// TwinCAT 3 PLC project TcoCoreExamples
// Title: TcoCoreExamples
// Company: Vortex.Library
// Author: Inxton
// ProjectVersion: 0.6.0.913
// ProgramVersion: 3.1.4024.12
// libraries:
//   Tc2_Standard, * (Beckhoff Automation GmbH)
//   Tc2_System, * (Beckhoff Automation GmbH)
//   Tc3_Module, * (Beckhoff Automation GmbH)
//   TcoCore, 0.6.0.913 (Vortex.Library)
// project tree:
//   Examples/Components/Digital/TcoDi/ TcoDi.TcPOU, TcoDiConfig.TcDUT
//   Examples/Components/Digital/TcoDo/ TcoDo.TcPOU
//   Examples/Components/ fbPiston.TcPOU, fbPistonConfig.TcDUT, fbPistonStatus.TcDUT, fbPistonMoveTask.TcPOU, IPistonGripper.TcIO, IPistonHorizontal.TcIO, IPistonVertical.TcIO
//   Examples/Components/WrappedComponent/ Example1WrappedComponent.TcPOU, Example2WrappedComponent.TcPOU, Example2WrappedComponents.TcDUT, Example2WrappedComponents_Status.TcDUT, Example2WrappedComponents_Config.TcDUT, Example2WrappedComponents_Control.TcDUT
//   Examples/Dialogs/ DiaglogsContext.TcPOU, MyOwnContent.TcPOU
//   Examples/ EXAMPLES_PRG.TcPOU, fbContext.TcPOU
//   Examples/Implementation/TcoContext/ TcoContext_App_1.TcPOU
//   Examples/Implementation/TcoObject/ TcoObject_Counter.TcPOU
//   Examples/Implementation/TcoState/ TcoContext_App_2.TcPOU
//   Examples/Implementation/TcoTask/ TcoTask_DownCounter.TcPOU
//   Examples/Logger/ LoggerContext.TcPOU, LoggerUsage.TcPOU
//   Examples/Manipulator/ fbManipulatorAutomat.TcPOU, fbManipulatorContext.TcPOU, gMANIPULATOR_IO.TcGVL, MANIPULATOR.TcPOU
//   Examples/Recorder/ RecordableStation001.TcPOU, RecordableStation001_Components.TcPOU, RecordableStation001_Sequencer.TcPOU
//   Examples/Station_001/ Station001.TcPOU, Station001_Components.TcPOU, Station001_Sequencer.TcPOU
//   Examples/Station_002/ Station002.TcPOU
//   Examples/Structured/ StructuredData.TcDUT, StructuredObject.TcPOU, StrucuredContext.TcPOU
//   Examples/WaveForm/ eTransitionType.TcDUT, TcoContext_Waveform.TcPOU, TcoObject_Waveform.TcPOU, TcoState_WaveformSequence.TcPOU, TcoTask_Transition.TcPOU, WaveformPoint.TcDUT
//   / PlcTask.TcTTO
//   POUs/ MAIN.TcPOU
// (motion and I/O tree: see PLC project tcocore)
// real-time tasks:
//   TASK PlcTask: cycle T#10ms, priority 20, ADS port 350
//   TASK PlcTask1: cycle T#10ms, priority 21, ADS port 351
//   TASK PlcTask2: cycle T#10ms, priority 22, ADS port 352

CONFIGURATION TcoCoreExamples
    RESOURCE PLC ON TwinCAT3
        TASK PlcTask(INTERVAL := T#10ms, PRIORITY := 22);
        PROGRAM MAIN WITH PlcTask : MAIN;
    END_RESOURCE
END_CONFIGURATION

// ---- Examples/Components/Digital/TcoDi/TcoDiConfig.TcDUT
TYPE TcoDiConfig :
STRUCT
    IsFalseTimeOut : TIME := T#10S;
    IsTrueTimeOut : TIME := T#10S;
END_STRUCT
END_TYPE

// ---- Examples/Components/fbPistonConfig.TcDUT
TYPE fbPistonConfig :
STRUCT
    MaxTimeToReachHome : TIME;
    MaxTimeToReachWork : TIME;
END_STRUCT
END_TYPE

// ---- Examples/Components/fbPistonStatus.TcDUT
TYPE fbPistonStatus :
STRUCT
    AtHome : TIME;
    AtWork : TIME;
END_STRUCT
END_TYPE

// ---- Examples/Components/WrappedComponent/Example2WrappedComponents.TcDUT
TYPE Example2WrappedComponents EXTENDS TcoCore.TcoStruct :
STRUCT
    {attribute addProperty Name "Pneumatic cyclinder"}
    piston : fbPiston(THISSTRUCT);
    digitalInput : TcoDi(THISSTRUCT);
    digitaOutput : TcoDo(THISSTRUCT);
    dummy1Task : TcoCore.TcoTask(THISSTRUCT);
    dummy2Task : TcoCore.TcoTask(THISSTRUCT);
    Setpoint : INT;
END_STRUCT
END_TYPE

// ---- Examples/Components/WrappedComponent/Example2WrappedComponents_Status.TcDUT
TYPE Example2WrappedComponents_Status EXTENDS TcoCore.TcoStruct :
STRUCT
    Feedback1 : INT;
    Feedback2 : BOOL;
    Feedback3 : STRING;
END_STRUCT
END_TYPE

// ---- Examples/Components/WrappedComponent/Example2WrappedComponents_Config.TcDUT
TYPE Example2WrappedComponents_Config EXTENDS TcoCore.TcoStruct :
STRUCT
    Setpoint1 : INT;
    Active : BOOL;
    FeedbackRequest : STRING;
END_STRUCT
END_TYPE

// ---- Examples/Components/WrappedComponent/Example2WrappedComponents_Control.TcDUT
TYPE Example2WrappedComponents_Control EXTENDS TcoCore.TcoStruct :
STRUCT
    Setpoint1 : INT;
    Up : BOOL;
    CommandAscii : STRING;
END_STRUCT
END_TYPE

// ---- Examples/Structured/StructuredData.TcDUT
TYPE StructuredData EXTENDS TcoCore.TcoStruct :
STRUCT
    _o1 :
STRUCTuredObject(THISSTRUCT);
END_STRUCT
END_TYPE

// ---- Examples/WaveForm/eTransitionType.TcDUT
{attribute 'qualified_only'}
{attribute 'strict'}
TYPE eTransitionType :
(
    None := 0,
    Linear := 1,
    Exponential := 2,
    S_Type := 3
);
END_TYPE

// ---- Examples/WaveForm/WaveformPoint.TcDUT
TYPE WaveformPoint :
STRUCT
    TransitionType : eTransitionType;
    TargetValue : LREAL; //Value to be reached in "Duration" PLC cycles
    Duration : UINT; //Number of PLC cycles during which the "TargetValue" must be reached
    Shape : LREAL; //Define curve shape
END_STRUCT
END_TYPE

// ---- Examples/Manipulator/gMANIPULATOR_IO.TcGVL
{attribute 'qualified_only'}
VAR_GLOBAL
    Inputs AT %I* : ARRAY[0..7] OF BOOL;
    Outputs AT %Q* : ARRAY[0..7] OF BOOL;
END_VAR

// ---- Examples/Components/IPistonGripper.TcIO
INTERFACE IPistonGripper

METHOD Close : TcoCore.ITcoTaskStatus
END_METHOD

METHOD Open : TcoCore.ITcoTaskStatus
END_METHOD

END_INTERFACE

// ---- Examples/Components/IPistonHorizontal.TcIO
INTERFACE IPistonHorizontal

METHOD MoveLeft : TcoCore.ITcoTaskStatus
END_METHOD

METHOD MoveRight : TcoCore.ITcoTaskStatus
END_METHOD

END_INTERFACE

// ---- Examples/Components/IPistonVertical.TcIO
INTERFACE IPistonVertical

METHOD MoveDown : TcoCore.ITcoTaskStatus
END_METHOD

METHOD MoveUp : TcoCore.ITcoTaskStatus
END_METHOD

END_INTERFACE

// ---- POUs/MAIN.TcPOU
PROGRAM MAIN
VAR
    _station001 : Station001;
    _station002 : Station002;
END_VAR

EXAMPLES_PRG();
MANIPULATOR();
_station001._sequence.DeactivateDeveloperChecks();
_station001.Run();
_station002.Run();

END_PROGRAM

// ---- Examples/Station_001/Station001.TcPOU
FUNCTION_BLOCK Station001 EXTENDS TcoCore.TcoContext
VAR
    {attribute addProperty Name "Long running example"}
    LongRunningTask : TcoCore.TcoTask(THIS^);
    i : int;
    _components : Station001_Components(THIS^);
    _sequence : Station001_Sequencer(THIS^, eRestoreMode.None, _components);
END_VAR

(*~
    <docu>
        <summary>
            Main method of the TcoContext. This is the entry point of any control logic that belongs to this context.
            The call of this method is ensured by calling the <c>InstanceName.Run()</c> method, and it must not be called explicitly.
            This method is abstract, and it must be overridden in derived block.
        </summary>
    </docu>
~*)
METHOD PROTECTED Main
_sequence.Run();

IF (LongRunningTask.Execute()) THEN
    i := i + 1;

    IF (i MOD 2000 = 0) THEN
        i := 1;
        LongRunningTask.DoneWhen(TRUE);
    END_IF
END_IF
END_METHOD

END_FUNCTION_BLOCK

// ---- Examples/Station_001/Station001_Components.TcPOU
FUNCTION_BLOCK Station001_Components EXTENDS TcoCore.TcoObject
VAR
    {attribute addProperty Name "Horizontal cyclinder A1"}
    _horizontal : fbPiston(THIS^);
    {attribute addProperty Name "Vertical cyclinder A2"}
    _vertical : fbPiston(THIS^);
    {attribute addProperty Name "Gripper A3"}
    _gripper : fbPiston(THIS^);
    {attribute addProperty Name "Digital input"}
    _di : TcoDi(THIS^);
    {attribute addProperty Name "Wrapped component example 1"}
    _wrappedComponent1 : Example1WrappedComponent(THIS^);
    {attribute addProperty Name "Wrapped component example 2"}
    _wrappedComponent2 : Example2WrappedComponent(THIS^);
    {attribute clr [RenderIgnore()]}
    _wrappedComponents : Example2WrappedComponents;
    tempSisgnal : BOOL;
    temp2Sisgnal : BOOL;
END_VAR
VAR
    _simTimerValue : UINT := 500;
    _simTimer : Tc2_Standard.TON;
END_VAR

_vertical();
_vertical.Service();
_horizontal();
_horizontal.Service();
_gripper();
_wrappedComponent1(inSignal := tempSisgnal);
_wrappedComponent1.Service();
_wrappedComponent2.Components.digitalInput(inoSignal := tempSisgnal);
_wrappedComponent2.Components.digitaOutput(inoSignal := temp2Sisgnal);
_wrappedComponent2();
_wrappedComponent2.Service();
_simTimer(IN := TRUE, PT := UINT_TO_TIME(_simTimerValue));
SimulateCylinder(_vertical);
SimulateCylinder(_horizontal);
SimulateCylinder(_gripper);

PROPERTY Gripper : IPistonGripper
GET
Gripper := _gripper;
END_GET
END_PROPERTY

PROPERTY Horizontal : IPistonHorizontal
GET
Horizontal := _horizontal;
END_GET
END_PROPERTY

METHOD SimulateCylinder
VAR_IN_OUT
    ioCyclinder : fbPiston;
END_VAR
ioCyclinder.iHomePositionSensor := ioCyclinder.qHomePositionActuator AND _simTimer.Q;
ioCyclinder.iWorkPositionSensor := ioCyclinder.qWorkPositionActuator AND _simTimer.Q;
END_METHOD

PROPERTY Vertical : IPistonVertical
GET
Vertical := _vertical;
END_GET
END_PROPERTY

END_FUNCTION_BLOCK

// ---- Examples/Components/fbPiston.TcPOU
{attribute addProperty Name "Pneumatic cyclinder"}
FUNCTION_BLOCK fbPiston EXTENDS TcoCore.TcoComponent IMPLEMENTS IPistonGripper, IPistonHorizontal, IPistonVertical
VAR_INPUT
    iHomePositionSensor : BOOL;
    iWorkPositionSensor : BOOL;
END_VAR
VAR_OUTPUT
    qHomePositionActuator : BOOL;
    qWorkPositionActuator : BOOL;
END_VAR
VAR
    {attribute addProperty Activity "moves to home position"}
    _moveHomeTask : fbPistonMoveTask(THIS^);
    {attribute addProperty Activity "moves to work position"}
    _moveWorkTask : fbPistonMoveTask(THIS^);
    _moveHomeMomentaryTask : TcoCore.TcoMomentaryTask(THIS^);
    _moveHomeToggleTask : TcoCore.TcoToggleTask(THIS^, FALSE);
    _config : fbPistonConfig;
    _status : fbPistonStatus;
END_VAR

_moveHomeTask(PositionSensor := iHomePositionSensor, MoveToPositionSignal := qHomePositionActuator, InverseSignal := qWorkPositionActuator);
_moveWorkTask(PositionSensor := iWorkPositionSensor, MoveToPositionSignal := qWorkPositionActuator, InverseSignal := qHomePositionActuator);
_moveHomeMomentaryTask.Run();
_moveHomeToggleTask.Toggle();

METHOD Close : TcoCore.ITcoTaskStatus
Close := MoveToHome();
END_METHOD

METHOD MoveDown : TcoCore.ITcoTaskStatus
MoveDown := MoveToHome();
END_METHOD

METHOD MoveLeft : TcoCore.ITcoTaskStatus
MoveLeft := MoveToWork();
END_METHOD

METHOD MoveRight : TcoCore.ITcoTaskStatus
MoveRight := MoveToHome();
END_METHOD

METHOD PROTECTED MoveToHome : TcoCore.ITcoTaskStatus
MoveToHome := THIS^._moveHomeTask.Invoke();
END_METHOD

METHOD PROTECTED MoveToWork : TcoCore.ITcoTaskStatus
MoveToWork := THIS^._moveWorkTask.Invoke();
END_METHOD

METHOD MoveUp : TcoCore.ITcoTaskStatus
MoveUp := MoveToWork();
END_METHOD

METHOD Open : TcoCore.ITcoTaskStatus
Open := MoveToWork();
END_METHOD

METHOD Restore : ITcoRestorable
THIS^._moveHomeTask.Restore();
THIS^._moveWorkTask.Restore();
END_METHOD

(*~
    <docu>
        <summary>
            Custom service (manual, maintenance) logic.
            This method must be implemented in derived class.
        </summary>
    </docu>
~*)
METHOD PROTECTED ServiceMode
END_METHOD

END_FUNCTION_BLOCK

// ---- Examples/Components/fbPistonMoveTask.TcPOU
{attribute addProperty Activity "task is running"}
FUNCTION_BLOCK fbPistonMoveTask EXTENDS TcoCore.TcoTask
VAR_INPUT
    PositionSensor : BOOL;
END_VAR
VAR_IN_OUT
    MoveToPositionSignal : BOOL;
    InverseSignal : BOOL;
END_VAR

IF (THIS^.Execute()) THEN
    THIS^.Messenger.Debug('|[[1]AttributeName]| |[AttributeActivity]|, extremity sensor not reached yet.');
    InverseSignal := FALSE;
    MoveToPositionSignal := TRUE;
    ThrowWhen(THIS^.ElapsedTime > T#5S);
    THIS^.DoneWhen(PositionSensor);
END_IF

END_FUNCTION_BLOCK

// ---- Examples/Components/Digital/TcoDi/TcoDi.TcPOU
(*~
    <docu>
        <summary>
                Generic component for monitoring of an input. (e.g. DigitalSensor).
        </summary>
    </docu>
~*)
FUNCTION_BLOCK TcoDi EXTENDS TcoCore.TcoComponent
VAR_IN_OUT
    (*~
    <docu>
        <summary>
            Input signal. Typically an `%I*` variable.
        </summary>
    </docu>
    ~*)
    inoSignal : BOOL;
END_VAR
VAR
    (*~
    <docu>
        <summary>
            Backing variable for signal; this variable is used directly by the component. It updates `inoSingal` in FB body call.
        </summary>
    </docu>
    ~*)
    _signal : BOOL;
END_VAR
VAR
    {attribute addProperty Name "<#Signal#>"}
    _signalInfo : TcoCore.TcoSignalInfo;
    {attribute addProperty Name "<#Check On#>"}
    {attribute addProperty ToolTip "<#Checks that the input is on#>"}
    _isTrueTask : TcoCore.TcoTask(THIS^);
    {attribute addProperty ToolTip "<#Checks that the input is off#>"}
    {attribute addProperty Name "<#Check Off#>"}
    _isFalseTask : TcoCore.TcoTask(THIS^);
    _config : TcoDiConfig;
    _isFalseTimeOutTimers : Tc2_Standard.TON;
    _isTrueTimeOutTimers : Tc2_Standard.TON;
END_VAR

IF (__ISVALIDREF(inoSignal)) THEN
    _signalInfo.GetSignalInfo(SIZEOF(inoSignal), ADR(inoSignal));
    _signal := inoSignal;
END_IF;

IF (_isTrueTask.Execute()) THEN
    _isTrueTask.DoneWhen(IsTrue);
END_IF

IF (_isFalseTask.Execute()) THEN
    _isFalseTask.DoneWhen(IsFalse);
END_IF

PROPERTY Config : REFERENCE TO TcoDiConfig
GET
Config REF= _config;
END_GET
END_PROPERTY

METHOD FB_init : BOOL
VAR_INPUT
    bInitRetains : BOOL; // if TRUE, the retain variables are initialized (warm start / cold start)
    bInCopyCode : BOOL; // if TRUE, the instance afterwards gets moved into the copy code (online change)
    ParentObject : ITcoObject;
END_VAR
END_METHOD

(*~
    <docu>
        <summary>
            Gets 'true' when monitor signal is 'off/false/logical 0'.
            Generates message when the returning 'false'.
        </summary>
    </docu>
~*)
{attribute 'monitoring' := 'variable'}
PROPERTY IsFalse : BOOL
GET
IsFalse := NOT _signal;
_isFalseTimeOutTimers(IN := NOT IsFalse, PT := _config.IsFalseTimeOut);

IF (NOT IsFalse) THEN
    Messenger.Info('<#Expecting `negative` signal#>');
END_IF;

IF (_isFalseTimeOutTimers.Q) THEN
    Messenger.Warning('<#Expecting `negative` signal#>');
END_IF;
END_GET
END_PROPERTY

(*~
    <docu>
        <summary>
            Gets 'true' when monitor signal is 'on/true/logical 1'.
            Generates message when the returning 'false'.
        </summary>
    </docu>
~*)
{attribute 'monitoring' := 'variable'}
PROPERTY IsTrue : BOOL
GET
IsTrue := _signal;
_isTrueTimeOutTimers(IN := NOT IsTrue, PT := _config.IsFalseTimeOut);

IF (NOT IsTrue) THEN
    Messenger.Info('<#Expecting `positive` signal#>');
END_IF;

IF (_isTrueTimeOutTimers.Q) THEN
    Messenger.Warning('<#Expecting `positive` signal#>');
END_IF;
END_GET
END_PROPERTY

(*~
    <docu>
        <summary>
            Restores this instance to the Ready state. Can be called explicitly or from within one of the restore mechanisms.
        </summary>
    </docu>
~*)
METHOD Restore : ITcoRestorable
// No implementation needed for this componet.
END_METHOD

(*~
    <docu>
        <summary>
            Custom service (manual, maintenance) logic.
            This method must be implemented in derived class.
        </summary>
    </docu>
~*)
METHOD PROTECTED ServiceMode
END_METHOD

PROPERTY PUBLIC Signal : Bool
GET
Signal := _signal;
END_GET
END_PROPERTY

END_FUNCTION_BLOCK

// ---- Examples/Components/WrappedComponent/Example1WrappedComponent.TcPOU
FUNCTION_BLOCK Example1WrappedComponent EXTENDS TcoCore.TcoComponent
VAR_INPUT
    inSignal : BOOL;
END_VAR
VAR_OUTPUT
END_VAR
VAR
    piston : fbPiston(THIS^);
    digitalInput : TcoDi(THIS^);
    digitaOutput : TcoDo(THIS^);
    dummy1Task : TcoCore.TcoTask(THIS^);
    dummy2Task : TcoCore.TcoTask(THIS^);
    Setpoint : INT;
END_VAR

piston();
digitalInput(inoSignal := inSignal);
dummy1Task.Enabled := TRUE;

IF dummy1Task.Execute() THEN
    ;
END_IF

(*~
    <docu>
        <summary>
            Restores this instance to the Ready state. Can be called explicitly or from within one of the restore mechanisms.
        </summary>
    </docu>
~*)
METHOD Restore : ITcoRestorable
END_METHOD

(*~
    <docu>
        <summary>
            Custom service (manual, maintenance) logic.
            This method must be implemented in derived class.
        </summary>
    </docu>
~*)
METHOD PROTECTED ServiceMode
piston.Service();
digitalInput.Service();
digitaOutput.Service();
END_METHOD

END_FUNCTION_BLOCK

// ---- Examples/Components/Digital/TcoDo/TcoDo.TcPOU
(*~
    <docu>
        <summary>
                Generic component for discrete control of an output.
        </summary>
    </docu>
~*)
FUNCTION_BLOCK TcoDo EXTENDS TcoCore.TcoComponent
VAR_IN_OUT
    (*~
    <docu>
        <summary>
            Controlled signal. Typically an `%Q*` variable.
        </summary>
    </docu>
    ~*)
    inoSignal : BOOL;
END_VAR
VAR
    (*~
    <docu>
        <summary>
            Backing variable for signal; this variable is used directly by the component. It updates `inoSingal` in FB body call.
        </summary>
    </docu>
    ~*)
    _signal : BOOL;
END_VAR
VAR
    {attribute addProperty Name "<#Signal#>"}
    _signalInfo : TcoCore.TcoSignalInfo;
    {attribute addProperty Name "<#On#>"}
    {attribute addProperty ToolTip "<#Sets the output#>"}
    _setTask : TcoCore.TcoTask(THIS^);
    {attribute addProperty ToolTip "<#Resets the output#>"}
    {attribute addProperty Name "<#Off#>"}
    _resetTask : TcoCore.TcoTask(THIS^);
END_VAR

IF (__ISVALIDREF(inoSignal)) THEN
    _signalInfo.GetSignalInfo(SIZEOF(inoSignal), ADR(inoSignal));
    inoSignal := _signal;
END_IF;

IF (_setTask.Execute()) THEN
    _setTask.DoneWhen(Set());
END_IF

IF (_resetTask.Execute()) THEN
    _resetTask.DoneWhen(Reset());
END_IF

METHOD FB_init : BOOL
VAR_INPUT
    bInitRetains : BOOL; // if TRUE, the retain variables are initialized (warm start / cold start)
    bInCopyCode : BOOL; // if TRUE, the instance afterwards gets moved into the copy code (online change)
    ParentObject : ITcoObject;
END_VAR
END_METHOD

(*~
    <docu>
        <summary>
            Gets 'true' when monitor signal is 'off/false/logical 0'.
            Generates message when the returning 'false'.
        </summary>
    </docu>
~*)
{attribute 'monitoring' := 'variable'}
PROPERTY IsFalse : BOOL
GET
IsFalse := NOT _signal;

IF (NOT IsFalse) THEN
    Messenger.Info('<#Expecting `negative` signal#>');
END_IF;
END_GET
END_PROPERTY

(*~
    <docu>
        <summary>
            Gets 'true' when monitor signal is 'on/true/logical 1'.
            Generates message when the returning 'false'.
        </summary>
    </docu>
~*)
{attribute 'monitoring' := 'variable'}
PROPERTY IsTrue : BOOL
GET
IsTrue := _signal;

IF (NOT IsTrue) THEN
    Messenger.Info('<#Expecting `positive` signal#>');
END_IF;
END_GET
END_PROPERTY

(*~
    <docu>
        <summary>
            Sets controlled signal into 'off/false/logical 0'.
        </summary>
    </docu>
~*)
METHOD Reset : BOOL
Messenger.Trace('<#Reseting signal (off/false)#>');
_signal := FALSE;
Reset := TRUE;
END_METHOD

(*~
    <docu>
        <summary>
            Restores this instance to the Ready state. Can be called explicitly or from within one of the restore mechanisms.
        </summary>
    </docu>
~*)
METHOD Restore : ITcoRestorable
// No implementation needed for this componet.
END_METHOD

(*~
    <docu>
        <summary>
            Custom service (manual, maintenance) logic.
            This method must be implemented in derived class.
        </summary>
    </docu>
~*)
METHOD PROTECTED ServiceMode
END_METHOD

(*~
    <docu>
        <summary>
            Sets controlled signal into 'on/true/logical 1'.
        </summary>
    </docu>
~*)
METHOD PUBLIC Set : BOOL
Messenger.Trace('<#Setting signal (on/true)#>');
_signal := TRUE;
Set := TRUE;
END_METHOD

PROPERTY PUBLIC Signal : Bool
GET
Signal := _signal;
END_GET
END_PROPERTY

END_FUNCTION_BLOCK

// ---- Examples/Components/WrappedComponent/Example2WrappedComponent.TcPOU
FUNCTION_BLOCK Example2WrappedComponent EXTENDS TcoCore.TcoComponent
VAR_OUTPUT
END_VAR
VAR
    _config : Example2WrappedComponents_Config;
    _status : Example2WrappedComponents_Status;
    _control : Example2WrappedComponents_Control;
    _components : Example2WrappedComponents := (Parent := THIS^);
    _resetTask : TcoCore.TcoTask(THIS^);
    _restoreTask : TcoCore.TcoTask(THIS^);
    Setpoint : INT;
    {attribute clr [RenderIgnore()]}
    SetpointDoNotRender : INT;
END_VAR

_resetTask();

PROPERTY Components : REFERENCE TO Example2WrappedComponents
GET
Components ref= _components;
END_GET
END_PROPERTY

(*~
    <docu>
        <summary>
            Restores this instance to the Ready state. Can be called explicitly or from within one of the restore mechanisms.
        </summary>
    </docu>
~*)
METHOD Restore : ITcoRestorable
END_METHOD

(*~
    <docu>
        <summary>
            Custom service (manual, maintenance) logic.
            This method must be implemented in derived class.
        </summary>
    </docu>
~*)
METHOD PROTECTED ServiceMode
_components.piston.Service();
_components.digitalInput.Service();
_components.digitaOutput.Service();
END_METHOD

END_FUNCTION_BLOCK

// ---- Examples/Station_001/Station001_Sequencer.TcPOU
FUNCTION_BLOCK Station001_Sequencer EXTENDS TcoCore.TcoSequencer
VAR
    components : REFERENCE TO Station001_Components;
END_VAR
VAR
    _switchToStep : BOOL;
    _failedToLoad : BOOL;
END_VAR
VAR
    _onStateChangeCount : LREAL;
    _sequenceCompleteCount : LREAL;
    _stepsPerSequence : LREAL;
END_VAR
VAR
    _stepIdChange : INT := 400;
    _stepsCountChange : BOOL := FALSE;
END_VAR

METHOD FB_init : BOOL
VAR_INPUT
    bInitRetains : BOOL; // if TRUE, the retain variables are initialized (warm start / cold start)
    bInCopyCode : BOOL; // if TRUE, the instance afterwards gets moved into the copy code (online change)
    ParentObject : ITcoObject;
    AutoRestoreMode : eRestoreMode;
    refComponents : REFERENCE TO Station001_Components;
END_VAR
Components REF= refComponents;
END_METHOD

METHOD Init
VAR_INPUT
END_VAR
components();
END_METHOD

(*~
    <docu>
        <summary>
            Main method of the sequener. Custom code needs to be placed here. The sequencer is executed by call of InstanceName.Run() method.
            This method is abstract, and it must be overridden in derived block.
        </summary>
    </docu>
~*)
METHOD PROTECTED Main : BOOL
Init();
THIS^.Messenger.Info('Stations one sequencer is running.');

IF (Step(100, TRUE, 'MOVE ALL CYLINDERS TO GROUND POSITION')) THEN
    //-----------------------------------------------------
    StepCompleteWhen(components.Vertical.MoveUp().Done AND_THEN components.Horizontal.MoveLeft().Done AND_THEN components.Gripper.Open().Done);
    //-----------------------------------------------------
END_IF

IF (Step(200, TRUE, 'MOVE VERTICAL CYLINDER DOWN')) THEN
    //-----------------------------------------------------
    StepCompleteWhen(components.Vertical.MoveDown().Done);
    //-----------------------------------------------------
END_IF

IF NOT _stepsCountChange THEN
    IF (Step(300, TRUE, 'CLOSE GRIPPER')) THEN
        //-----------------------------------------------------
        IF (components.Gripper.Close().Done) THEN
            IF (_failedToLoad) THEN
                RequestStep(100);
            ELSE
                StepCompleteWhen(TRUE);
            END_IF;
        END_IF;
        //-----------------------------------------------------
    END_IF

    IF (Step(_stepIdChange, TRUE, 'MOVE VERTICAL CYLINDER UP')) THEN
        //-----------------------------------------------------
        StepCompleteWhen(components.Vertical.MoveUp().Done);
        //-----------------------------------------------------
    END_IF

    IF (Step(500, TRUE, 'MOVE HORIZONTAL CYLINDER TO UNLOAD POSITION')) THEN
        //-----------------------------------------------------
        StepCompleteWhen(components.Horizontal.MoveRight().Done);
        //-----------------------------------------------------
    END_IF
END_IF

IF (Step(600, TRUE, 'MOVE VERTICAL CYLINDER DOWN')) THEN
    //-----------------------------------------------------
    StepCompleteWhen(components.Vertical.MoveDown().Done);
    //-----------------------------------------------------
END_IF

IF (Step(700, TRUE, 'OPEN GRIPPER')) THEN
    //-----------------------------------------------------
    StepCompleteWhen(components.Gripper.Open().Done);
    //-----------------------------------------------------
END_IF

IF (Step(800, TRUE, 'CLOSE SEQUENCE')) THEN
    //-----------------------------------------------------
    _sequenceCompleteCount := _sequenceCompleteCount + 1;
    _stepsPerSequence := (_onStateChangeCount - _sequenceCompleteCount + 1) / _sequenceCompleteCount;
    CompleteSequence();
    //-----------------------------------------------------
END_IF

THIS^.Messenger.Debug('THIS IS DEBUG DIAG MESSAGE ');
THIS^.Messenger.Info('THIS IS INFO DIAG MESSAGE ');
THIS^.Messenger.Notify('THIS IS NOTIFY DIAG MESSAGE ');
THIS^.Messenger.Warning('THIS IS WARNING DIAG MESSAGE ');
//THIS^.Messenger.Error('THIS IS ERROR DIAG MESSAGE ');
//THIS^.Messenger.Programming('THIS IS PROGRAMMING DIAG MESSAGE ');
//THIS^.Messenger.Post('THIS IS Fatal DIAG MESSAGE ', eMessageCategory.Fatal);
//THIS^.Messenger.Post('THIS IS Critical DIAG MESSAGE ', eMessageCategory.Critical);
//THIS^.Messenger.Post('THIS IS Catastrophic DIAG MESSAGE ', eMessageCategory.Catastrophic);
THIS^.Messenger.Trace('THIS IS INFO DIAG MESSAGE ');
END_METHOD

METHOD PROTECTED OnStateChange
VAR_INPUT
    PreviousState : INT;
    NewState : INT;
END_VAR
VAR
    sb : TcoCore.StringBuilder;
END_VAR
THIS^.Messenger.Trace(INT_TO_STRING(PreviousState));
_onStateChangeCount := _onStateChangeCount + 1;
components._simTimer(IN := FALSE);
END_METHOD

END_FUNCTION_BLOCK

// ---- Examples/Station_002/Station002.TcPOU
FUNCTION_BLOCK Station002 EXTENDS TcoCore.TcoContext
VAR
    {attribute addProperty Name "Horizontal cyclinder A1"}
    _horizontal : fbPiston(THIS^);
    {attribute addProperty Name "Vertical cyclinder A2"}
    _vertical : fbPiston(THIS^);
    {attribute addProperty Name "Gripper A3"}
    _gripper : fbPiston(THIS^);
END_VAR
VAR
    _s : TcoCore.TcoSequence(THIS^, eRestoreMode.None);
    _sObserver : TcoCore.TcoSequencerObserver(THIS^);
    _failedToLoad : BOOL;
END_VAR

(*~
    <docu>
        <summary>
            Main method of the TcoContext. This is the entry point of any control logic that belongs to this context.
            The call of this method is ensured by calling the <c>InstanceName.Run()</c> method, and it must not be called explicitly.
            This method is abstract, and it must be overridden in derived block.
        </summary>
    </docu>
~*)
METHOD PROTECTED Main
_s.Open();
THIS^._s.Observer := _sObserver;
THIS^._s.Messenger.Info('Stations two sequencer is running.');

IF (_s.Step(100, TRUE, 'MOVE ALL CYLINDERS TO GROUND POSITION')) THEN
    //-----------------------------------------------------
    _s.StepCompleteWhen(_vertical.MoveUp().Done AND_THEN _horizontal.MoveLeft().Done AND_THEN _gripper.Open().Done);
    //-----------------------------------------------------
END_IF

IF (_s.Step(200, TRUE, 'MOVE VERTICAL CYLINDER DOWN')) THEN
    //-----------------------------------------------------
    _s.StepCompleteWhen(_vertical.MoveDown().Done);
    //-----------------------------------------------------
END_IF

IF (_s.Step(300, TRUE, 'CLOSE GRIPPER')) THEN
    //-----------------------------------------------------
    IF (_gripper.Close().Done) THEN
        IF (_failedToLoad) THEN
            _s.RequestStep(100);
        ELSE
            _s.StepCompleteWhen(TRUE);
        END_IF;
    END_IF;
    //-----------------------------------------------------
END_IF

IF (_s.Step(400, TRUE, 'MOVE VERTICAL CYLINDER UP')) THEN
    //-----------------------------------------------------
    _s.StepCompleteWhen(_vertical.MoveUp().Done);
    //-----------------------------------------------------
END_IF

IF (_s.Step(500, TRUE, 'MOVE HORIZONTAL CYLINDER TO UNLOAD POSITION')) THEN
    //-----------------------------------------------------
    _s.StepCompleteWhen(_horizontal.MoveRight().Done);
    //-----------------------------------------------------
END_IF

IF (_s.Step(600, TRUE, 'MOVE VERTICAL CYLINDER DOWN')) THEN
    //-----------------------------------------------------
    _s.StepCompleteWhen(_vertical.MoveDown().Done);
    //-----------------------------------------------------
END_IF

IF (_s.Step(700, TRUE, 'OPEN GRIPPER')) THEN
    //-----------------------------------------------------
    _s.StepCompleteWhen(_gripper.Open().Done);
    //-----------------------------------------------------
END_IF

IF (_s.Step(800, TRUE, 'CLOSE SEQUENCE')) THEN
    //-----------------------------------------------------
    _s.CompleteSequence();
    //-----------------------------------------------------
END_IF

_s.Close();
END_METHOD

END_FUNCTION_BLOCK

// ---- Examples/EXAMPLES_PRG.TcPOU
PROGRAM EXAMPLES_PRG
VAR
    _context : fbContext;
    _recordableStations : RecordableStation001;
    _loggerContext : LoggerContext;
    _strucuredContext : StrucuredContext;
    _diaglogsContext : DiaglogsContext;
    a : TcoCore.ITcoObject;
END_VAR

_context.Run();
_recordableStations.Run();
_loggerContext.Run();
_diaglogsContext.Run();
a := _strucuredContext._structuredData._o1.Parent;

END_PROGRAM

// ---- Examples/fbContext.TcPOU
FUNCTION_BLOCK fbContext EXTENDS TcoCore.TcoContext
VAR
    {attribute addProperty Name "Toggle task example"}
    {attribute addProperty StateOnDesc "<#Enabled#>"}
    {attribute addProperty StateOffDesc "<#Disabled#>"}
    _toggleTaskExample : TcoCore.TcoToggleTask(THIS^, FALSE);
    {attribute addProperty Name "Momentary task example"}
    {attribute addProperty StateOnDesc "<#Running#>"}
    {attribute addProperty StateOffDesc "<#Stopped#>"}
    _momentaryTaskExample : TcoCore.TcoMomentaryTask(THIS^);
END_VAR

METHOD PROTECTED Main
_toggleTaskExample.Run();
_momentaryTaskExample.Run();
END_METHOD

END_FUNCTION_BLOCK

// ---- Examples/Recorder/RecordableStation001.TcPOU
FUNCTION_BLOCK RecordableStation001 EXTENDS TcoCore.TcoContext
VAR
    _components : RecordableStation001_Components(THIS^);
    _sequence : RecordableStation001_Sequencer(THIS^, eRestoreMode.None);
    _serviceModeTask : TcoCore.TcoTask(THIS^);
    _automatModeTask : TcoCore.TcoTask(THIS^);
END_VAR

(*~
    <docu>
        <summary>
            Main method of the TcoContext. This is the entry point of any control logic that belongs to this context.
            The call of this method is ensured by calling the <c>InstanceName.Run()</c> method, and it must not be called explicitly.
            This method is abstract, and it must be overridden in derived block.
        </summary>
    </docu>
~*)
METHOD PROTECTED Main
_sequence(components := _components);
_components();

IF (_serviceModeTask.Execute()) THEN
    _automatModeTask.Restore();
    _components.Service();
END_IF;

IF (_automatModeTask.Execute()) THEN
    _serviceModeTask.Restore();
    _sequence.Run();
END_IF;
END_METHOD

END_FUNCTION_BLOCK

// ---- Examples/Recorder/RecordableStation001_Components.TcPOU
FUNCTION_BLOCK RecordableStation001_Components EXTENDS TcoCore.TcoObject
VAR
    {attribute addProperty Name "Horizontal cyclinder A1"}
    _horizontal : fbPiston(THIS^);
    {attribute addProperty Name "Vertical cyclinder A2"}
    _vertical : fbPiston(THIS^);
    {attribute addProperty Name "Gripper A3"}
    _gripper : fbPiston(THIS^);
END_VAR
VAR
    _simTimerValue : UINT := 500;
    _simTimer : Tc2_Standard.TON;
END_VAR

_vertical();
_horizontal();
_gripper();

PROPERTY Gripper : IPistonGripper
GET
Gripper := _gripper;
END_GET
END_PROPERTY

PROPERTY Horizontal : IPistonHorizontal
GET
Horizontal := _horizontal;
END_GET
END_PROPERTY

METHOD Service
VAR_INPUT
END_VAR
THIS^._gripper.Service();
THIS^._horizontal.Service();
THIS^._vertical.Service();
END_METHOD

PROPERTY Vertical : IPistonVertical
GET
Vertical := _vertical;
END_GET
END_PROPERTY

END_FUNCTION_BLOCK

// ---- Examples/Recorder/RecordableStation001_Sequencer.TcPOU
FUNCTION_BLOCK RecordableStation001_Sequencer EXTENDS TcoCore.TcoSequencer
VAR_IN_OUT
    components : RecordableStation001_Components;
END_VAR
VAR
    _switchToStep : BOOL;
    _failedToLoad : BOOL;
END_VAR
VAR
    _onStateChangeCount : LREAL;
    _sequenceCompleteCount : LREAL;
    _stepsPerSequence : LREAL;
END_VAR

METHOD FB_init : BOOL
VAR_INPUT
    bInitRetains : BOOL; // if TRUE, the retain variables are initialized (warm start / cold start)
    bInCopyCode : BOOL; // if TRUE, the instance afterwards gets moved into the copy code (online change)
    ParentObject : ITcoObject;
    AutoRestoreMode : eRestoreMode;
END_VAR
END_METHOD

METHOD Init
VAR_INPUT
END_VAR
components();
END_METHOD

(*~
    <docu>
        <summary>
            Main method of the sequener. Custom code needs to be placed here. The sequencer is executed by call of InstanceName.Run() method.
            This method is abstract, and it must be overridden in derived block.
        </summary>
    </docu>
~*)
METHOD PROTECTED Main : BOOL
Init();

IF Step(10, TRUE, 'EXAMPLES_PRG._recordableStations._components._horizontal._moveHomeTask') THEN
    //-------------------------------------------------------
    IF (EXAMPLES_PRG._recordableStations._components._horizontal._moveHomeTask.Invoke().Done) THEN
        StepCompleteWhen(TRUE);
    END_IF;
    //-------------------------------------------------------
END_IF;

IF Step(20, TRUE, 'EXAMPLES_PRG._recordableStations._components._vertical._moveHomeTask') THEN
    //-------------------------------------------------------
    IF (EXAMPLES_PRG._recordableStations._components._vertical._moveHomeTask.Invoke().Done) THEN
        StepCompleteWhen(TRUE);
    END_IF;
    //-------------------------------------------------------
END_IF;

IF Step(30, TRUE, 'EXAMPLES_PRG._recordableStations._components._gripper._moveHomeTask') THEN
    //-------------------------------------------------------
    IF (EXAMPLES_PRG._recordableStations._components._gripper._moveHomeTask.Invoke().Done) THEN
        StepCompleteWhen(TRUE);
    END_IF;
    //-------------------------------------------------------
END_IF;
END_METHOD

METHOD PROTECTED OnStateChange
VAR_INPUT
    PreviousState : INT;
    NewState : INT;
END_VAR
_onStateChangeCount := _onStateChangeCount + 1;
components._simTimer(IN := FALSE);
END_METHOD

END_FUNCTION_BLOCK

// ---- Examples/Logger/LoggerContext.TcPOU
FUNCTION_BLOCK LoggerContext EXTENDS TcoCore.TcoContext
VAR
    _loggerUsage : LoggerUsage(THIS^);
END_VAR

(*~
    <docu>
        <summary>
            Main method of the TcoContext. This is the entry point of any control logic that belongs to this context.
            The call of this method is ensured by calling the <c>InstanceName.Run()</c> method, and it must not be called explicitly.
            This method is abstract, and it must be overridden in derived block.
        </summary>
    </docu>
~*)
METHOD PROTECTED Main
_loggerUsage();
END_METHOD

END_FUNCTION_BLOCK

// ---- Examples/Logger/LoggerUsage.TcPOU
FUNCTION_BLOCK LoggerUsage EXTENDS TcoCore.TcoObject
VAR
    _logger : TcoCore.TcoLogger(THIS^);
    _counter : INT;
END_VAR

//_counter := _counter + 1;
//IF((_counter MOD 100) = 0) THEN
//	_logger.Push('hey friend! we got a problem', eMessageCategory.Critical);
//END_IF;

END_FUNCTION_BLOCK

// ---- Examples/Structured/StrucuredContext.TcPOU
FUNCTION_BLOCK StrucuredContext EXTENDS TcoCore.TcoContext
VAR
    _structuredData :
STRUCTuredData := (Parent := THIS^);
END_VAR

(*~
    <docu>
        <summary>
            Main method of the TcoContext. This is the entry point of any control logic that belongs to this context.
            The call of this method is ensured by calling the <c>InstanceName.Run()</c> method, and it must not be called explicitly.
            This method is abstract, and it must be overridden in derived block.
        </summary>
    </docu>
~*)
METHOD PROTECTED Main
END_METHOD

END_FUNCTION_BLOCK

// ---- Examples/Dialogs/DiaglogsContext.TcPOU
FUNCTION_BLOCK DiaglogsContext EXTENDS TcoCore.TcoContext
VAR
    _invokeDiaglog1 : BOOL;
    _dialog1 : TcoCore.TcoDialog(THIS^);
    _dialog2 : TcoCore.TcoDialog(THIS^);
    _dialog3 : TcoCore.TcoDialog(THIS^);
    _dialog4 : TcoCore.TcoDialog(THIS^);
    _invokeDiaglogsConsequential : BOOL;
    _dialog1Consequential : TcoCore.TcoDialog(THIS^);
    _dialog2Consequential : TcoCore.TcoDialog(THIS^);
    _dialog3Consequential : TcoCore.TcoDialog(THIS^);
    diag : ITcoDialogAnswer;
    _tonDisposeDialog : TON;
    _state : INT;
    _invokeCustomizedDiaglog : BOOL;
    _dialogCustomized : TcoCore.TcoCustomizedDialog(THIS^);
    _invokeInputDiaglog : BOOL;
    _customizedContentInput : MyOwnContent(THIS^);
    _dialogWithInput : TcoCore.TcoInputDialog(THIS^);
END_VAR

(*~
    <docu>
        <summary>
            Main method of the TcoContext. This is the entry point of any control logic that belongs to this context.
            The call of this method is ensured by calling the <c>InstanceName.Run()</c> method, and it must not be called explicitly.
            This method is abstract, and it must be overridden in derived block.
        </summary>
    </docu>
~*)
METHOD PROTECTED Main
VAR
END_VAR
CASE _state OF
    0:
        _dialog1.Restore();
        _dialog2.Restore();
        _dialog3.Restore();
        _dialog4.Restore();
        _dialogWithInput.Restore();
        _dialogCustomized.Restore();

        IF (_invokeDiaglog1) THEN
            _state := 10;
        ELSIF (_invokeCustomizedDiaglog) THEN
            _state := 50;
        ELSIF (_invokeInputDiaglog) THEN
            _state := 100;
        END_IF;
    10:
        _dialog1.Show()
            .WithType(eDialogType.Question)
            .WithYesNoCancel()
            .WithImage('D:\MTS\Develop\TcOpenGroup\TcOpen\assets\logo\TcOpenLogo.png', 500, 500)
            .WithCaption('Hey 1').WithText('Do we go ahead to 2?');

        IF (_dialog1.Answer = TcoCore.eDialogAnswer.Yes) THEN
            _state := 15;
        END_IF;

        IF (_dialog1.Answer = TcoCore.eDialogAnswer.No) THEN
            _state := 1000;
        END_IF;

        IF (_dialog1.Answer = TcoCore.eDialogAnswer.Cancel) THEN
            _state := 0;
            _invokeDiaglog1 := FALSE;
        END_IF;
    15:
        _dialog1.Show().WithType(eDialogType.Question).WithYesNoCancel().WithImage('', 500, 500).WithCaption('Hey 2').WithText('Do we go ahead?');

        IF (_dialog1.Answer = TcoCore.eDialogAnswer.Yes) THEN
            _state := 20;
        END_IF;

        IF (_dialog1.Answer = TcoCore.eDialogAnswer.No) THEN
            _state := 1000;
        END_IF;

        IF (_dialog1.Answer = TcoCore.eDialogAnswer.Cancel) THEN
            _state := 0;
            _invokeDiaglog1 := FALSE;
        END_IF;
    20:
        IF (_dialog2.Show().WithType(eDialogType.Info).WithOk().WithCaption('Hey').WithText('We go ahead.').Answer = TcoCore.eDialogAnswer.OK) THEN
            _state := 30;
        END_IF
    30:
        _state := 40;
        _tonDisposeDialog(In := FALSE);
    40:
        _tonDisposeDialog(IN := TRUE, PT := T#4S);

        _dialog4.ShowWithExternalClose(inOkAnswerSignal := FALSE,
            inYesAnswerSignal := _tonDisposeDialog.Q,
            inNoAnswerSignal := FALSE,
            inCancelAnswerSignal := FALSE)
            .WithType(eDialogType.Info)
            .WithYesNoCancel()
            .WithCaption('Hey').WithText('Do you wana retry it? Yes answer will be set in 4 sec?');

        IF (_dialog4.Answer = TcoCore.eDialogAnswer.Yes) THEN
            _state := 0;
        END_IF;

        IF (_dialog4.Answer = TcoCore.eDialogAnswer.No) THEN
            _state := 50;
        END_IF;

        IF (_dialog4.Answer = TcoCore.eDialogAnswer.Cancel) THEN
            _state := 0;
            _invokeDiaglog1 := FALSE;
        END_IF;
    50:
        _dialogCustomized.Show()
            .WithType(eDialogType.Info)
            .WithOption1('This is Option1=>retry')
            .WithOption2('This is Option2=>first step')
            .WithOption3('This is Option3 =>continue')
            .WithOption4('This is Option4=>stop sequence')
            .WithCaption('Hey').WithText('What we are going to do.');

        IF (_dialogCustomized.Answer = TcoCore.eCustomizedDialogAnswer.Option1) THEN
            _state := 50;
        END_IF;

        IF (_dialogCustomized.Answer = TcoCore.eCustomizedDialogAnswer.Option2) THEN
            _state := 0;
        END_IF;

        IF (_dialogCustomized.Answer = TcoCore.eCustomizedDialogAnswer.Option3) THEN
            _state := 51;
        END_IF;

        IF (_dialogCustomized.Answer = TcoCore.eCustomizedDialogAnswer.Option4) THEN
            _state := 0;
            _invokeCustomizedDiaglog := FALSE;
            _invokeDiaglog1 := FALSE;
        END_IF;
    51:
        _dialogCustomized.Show()
            .WithOption1('This is Option1=>retry')
            .WithOption2('This is Option2=>first step')
            .WithOption3('This is Option3 =>continue')
            .WithImage('D:\MTS\Develop\TcOpenGroup\TcOpen\assets\logo\TcOpenWide.png', 500, 500)
            .WithCaption('Hey').WithText('What we are going to do.');

        IF (_dialogCustomized.Answer = TcoCore.eCustomizedDialogAnswer.Option1) THEN
            _state := 50;
        END_IF;

        IF (_dialogCustomized.Answer = TcoCore.eCustomizedDialogAnswer.Option2) THEN
            _state := 0;
        END_IF;

        IF (_dialogCustomized.Answer = TcoCore.eCustomizedDialogAnswer.Option3) THEN
            _state := 60;
        END_IF;

        IF (_dialogCustomized.Answer = TcoCore.eCustomizedDialogAnswer.Option4) THEN
            _state := 0;
            _invokeCustomizedDiaglog := FALSE;
            _invokeDiaglog1 := FALSE;
        END_IF;
    60:
        _state := 70;
        _tonDisposeDialog(In := FALSE);
    70:
        _tonDisposeDialog(IN := TRUE, PT := T#4S);

        _dialog4.ShowWithExternalClose(inOkAnswerSignal := FALSE,
            inYesAnswerSignal := _tonDisposeDialog.Q,
            inNoAnswerSignal := FALSE,
            inCancelAnswerSignal := FALSE)
            .WithType(eDialogType.Info)
            .WithYesNoCancel()
            .WithCaption('Hey').WithText('Do you wana retry it? Yes answer will be set in 4 sec?');

        IF (_dialog4.Answer = TcoCore.eDialogAnswer.Yes) THEN
            _state := 0;
        END_IF;

        IF (_dialog4.Answer = TcoCore.eDialogAnswer.No) THEN
            _state := 80;
        END_IF;

        IF (_dialog4.Answer = TcoCore.eDialogAnswer.Cancel) THEN
            _state := 0;
            _invokeDiaglog1 := FALSE;
        END_IF;
    80:
        _state := 90;
        _tonDisposeDialog(In := FALSE);
    90:
        _tonDisposeDialog(IN := TRUE, PT := T#4S);

        _dialogCustomized.ShowWithExternalClose(inOption1AnswerSignal := FALSE,
            inOption2AnswerSignal := FALSE,
            inOption3AnswerSignal := _tonDisposeDialog.Q,
            inOption4AnswerSignal := FALSE)
            .WithOption1('This is Option1=>retry')
            .WithOption2('This is Option2=>first step')
            .WithOption3('This is Option3 =>continue and finish in 4s')
            .WithImage('D:\MTS\Develop\TcOpenGroup\TcOpen\assets\logo\TcOpenWide.png', 500, 500)
            .WithCaption('Hey').WithText('What we are going to do.');

        IF (_dialogCustomized.Answer = TcoCore.eCustomizedDialogAnswer.Option1) THEN
            _state := 80;
        END_IF;

        IF (_dialogCustomized.Answer = TcoCore.eCustomizedDialogAnswer.Option2) THEN
            _state := 10;
        END_IF;

        IF (_dialogCustomized.Answer = TcoCore.eCustomizedDialogAnswer.Option3) THEN
            _state := 0;
            _invokeCustomizedDiaglog := FALSE;
            _invokeDiaglog1 := FALSE;
        END_IF;
    100:
        _dialogWithInput.Show(refContent := _customizedContentInput).WithType(eDialogType.Question).WithYesNo().WithCaption('Hey wana set data')
            .WithText('Do you realy want to sent data to ....?');

        IF (_dialogWithInput.Answer = TcoCore.eInputDialogAnswer.Yes) THEN
            _state := 110;
        END_IF;

        IF (_dialogWithInput.Answer = TcoCore.eInputDialogAnswer.No) THEN
            _invokeInputDiaglog := FALSE;
            _state := 1000;
        END_IF;
    110:
        _dialogWithInput.Show(refContent := _customizedContentInput)
            .WithType(eDialogType.Question)
            .WithOk()
            .WithImage('https://github.com/TcOpenGroup', 400, 600)
            .WithCaption('Hey wana set data').WithText('Do you realy want to sent data to ....?');

        IF (_dialogWithInput.Answer = TcoCore.eInputDialogAnswer.OK) THEN
            _state := 1000;
            _invokeInputDiaglog := FALSE;
        END_IF;
    1000:
        IF (_dialog3.Show().WithType(eDialogType.Warning).WithOk().WithCaption('Hey').WithText('We are done.').Answer = TcoCore.eDialogAnswer.OK)
            THEN
            _state := 0;
        END_IF
END_CASE

//IF(_invokeDiaglog1) THEN
//	IF(_dialog1.Answer = TcoCore.eDialogAnswer.Yes) THEN
//		IF(_dialog2.Show()
//			.WithType(eDialogType.Info)
//			.WithOk()
//			.WithCaption('Hey')
//			.WithText('We go ahead.')
//			.Answer = TcoCore.eDialogAnswer.OK) THEN
//			_invokeDiaglog1 := FALSE;
//		END_IF
//	ELSIF(_dialog1.Answer = TcoCore.eDialogAnswer.No) THEN
//		IF(_dialog3.Show()
//				  	.WithOk()
//					.WithCaption('Hey')
//					.WithText('We don`t go ahead.')
//					.Answer = TcoCore.eDialogAnswer.OK) THEN
//			_invokeDiaglog1 := FALSE;
//		END_IF
//	END_IF
//END_IF;
IF (_invokeDiaglogsConsequential) THEN
    _dialog1Consequential.Show().WithYesNoCancel().WithCaption('Hey D1').WithText('D1');
    _dialog2Consequential.Show().WithYesNoCancel().WithCaption('Hey D2').WithText('D2');
    _dialog3Consequential.Show().WithYesNoCancel().WithCaption('Hey D3').WithText('D3');
END_IF;
END_METHOD

END_FUNCTION_BLOCK

// ---- Examples/Dialogs/MyOwnContent.TcPOU
FUNCTION_BLOCK MyOwnContent EXTENDS TcoCore.TcoInputDialogContentContainer
VAR_INPUT
END_VAR
VAR_OUTPUT
END_VAR
VAR
    {attribute addProperty Name "<#Recipe#>"}
    Recipe : STRING;
    {attribute addProperty Name "<#Qantity#>"}
    RequiredQuantity : INT;
    {attribute addProperty Name "<#Timeout#>"}
    Timeout : DATE_AND_TIME;
    {attribute addProperty Name "<#Exclude#>"}
    Exclude : BOOL;
END_VAR

END_FUNCTION_BLOCK

// ---- Examples/Manipulator/MANIPULATOR.TcPOU
PROGRAM MANIPULATOR
VAR
    _context : fbManipulatorContext;
END_VAR

_context.Run();

END_PROGRAM

// ---- Examples/Manipulator/fbManipulatorContext.TcPOU
FUNCTION_BLOCK fbManipulatorContext EXTENDS TcoCore.TcoContext
VAR
    _automat : fbManipulatorAutomat(THIS^, eRestoreMode.AutoRestoreMembers);
END_VAR

METHOD PROTECTED Main
_automat();
END_METHOD

END_FUNCTION_BLOCK

// ---- Examples/Manipulator/fbManipulatorAutomat.TcPOU
FUNCTION_BLOCK fbManipulatorAutomat EXTENDS TcoCore.TcoState
VAR
    _horizontalPiston : fbPiston(THIS^);
    _verticalPiston : fbPiston(THIS^);
    _gripperPiston : fbPiston(THIS^);
    _persistentMessage : TcoCore.TcoMessenger(THIS^);
END_VAR
VAR
    ar : ARRAY[0..2] OF BOOL;
END_VAR
VAR
    _bool : BOOL;
    _real : REAL := 1.5;
    _lreal : LREAL := 2.5;
    _dt : DT := DT#2013-05-09-13:29:20.500;
    _d : DATE := D#2012-04-14;
    _time : TIME := T#50MS;
    _string : STRING := 'str';
    _wstring : WSTRING := "wstr";
    _tod : TOD := TOD#13:29:20.500;
    _int : INT := 589;
END_VAR

// THIS^.Context.Environment.Messaging.Suspend();
_persistentMessage.OnCondition(TRUE)
    .Build() //.Append('sss').Append('ddd')
//.AppendAny(ar[0])
    .AppendAny(_bool)
    .AppendAny(_real)
    .AppendAny(_lreal)
    .AppendAny(_dt)
    .AppendAny(_d)
    .AppendAny(_time)
    .AppendAny(_string)
    .AppendAny(_wstring)
    .AppendAny(_tod)
    .AppendAny(_int)
    .As().AsDebug();

IF (NOT _persistentMessage.OnCondition(ar[0]).Build().Append('This is problem ').Append('like any other').As().AsError().Pin().Pinned) THEN
    _persistentMessage.OnCondition(ar[1]).Error('this is persistent error 2').Pin();
END_IF;

IF (ar[2]) THEN
    _persistentMessage.UnPin();
END_IF;

RETURN;

THIS^._verticalPiston.Messenger
    .OnCondition(THIS^.Context.StartCycleCount MOD 5000 = 0)
    .Post('We are running automatic mode4 conditional', eMessageCategory.Catastrophic).Pin();

THIS^.Messenger.OnCondition(THIS^.Context.StartCycleCount MOD 2500 = 0).Info('We are running automatic mode1 conditional').Pin();
THIS^._gripperPiston.Messenger.OnCondition(THIS^.Context.StartCycleCount MOD 1000 = 0).Notify('We are running automatic mode7 conditional').Pin();
//IF(THIS^.Context.StartCycleCount MOD 1 = 0) THEN
THIS^.Messenger.Info('We are running automatic mode1');
THIS^.Messenger.Notify('We are running automatic mode2');
THIS^.Messenger.Notify('We are running automatic mode3');
THIS^._verticalPiston.Messenger.Notify('We are running automatic mode4');
THIS^._verticalPiston.Messenger.Notify('We are running automatic mode5');
THIS^._verticalPiston.Messenger.Notify('We are running automatic mode6');
THIS^._gripperPiston.Messenger.Notify('We are running automatic mode7');
THIS^._gripperPiston.Messenger.Notify('We are running automatic mode8');
THIS^._gripperPiston.Messenger.Notify('We are running automatic mode9');
THIS^.Messenger.Info('We are running automatic mode1');
THIS^.Messenger.Notify('We are running automatic mode2');
THIS^.Messenger.Notify('We are running automatic mode3');
THIS^._verticalPiston.Messenger.Notify('We are running automatic mode4-');
THIS^._verticalPiston.Messenger.Notify('We are running automatic mode5-');
THIS^._verticalPiston.Messenger.Notify('We are running automatic mode6-');
THIS^._gripperPiston.Messenger.Notify('We are running automatic mode7-');
THIS^._gripperPiston.Messenger.Notify('We are running automatic mode8-');
THIS^._gripperPiston.Messenger.Notify('We are running automatic mode9-');
THIS^.Messenger.Info('We are running automatic mode1-');
THIS^.Messenger.Notify('We are running automatic mode2-');
THIS^.Messenger.Notify('We are running automatic mode3-');
THIS^._verticalPiston.Messenger.Notify('We are running automatic mode48');
THIS^._verticalPiston.Messenger.Notify('We are running automatic mode5');
THIS^._verticalPiston.Messenger.Notify('We are running automatic mode6');
THIS^._gripperPiston.Messenger.Notify('We are running automatic mode7');
THIS^._gripperPiston.Messenger.Notify('We are running automatic mode8');
THIS^._gripperPiston.Messenger.Notify('We are running automatic mode9');
THIS^.Messenger.Info('We are running automatic mode1');
THIS^.Messenger.Notify('We are running automatic mode2');
THIS^.Messenger.Notify('We are running automatic mode3');
THIS^._verticalPiston.Messenger.Notify('We are running automatic mode4');
THIS^._verticalPiston.Messenger.Notify('We are running automatic mode5');
THIS^._verticalPiston.Messenger.Notify('We are running automatic mode6');
THIS^._gripperPiston.Messenger.Notify('We are running automatic mode7');
THIS^._gripperPiston.Messenger.Notify('We are running automatic mode8');
THIS^._gripperPiston.Messenger.Notify('We are running automatic mode9');
THIS^.Messenger.Info('We are running automatic mode1');
THIS^.Messenger.Notify('We are running automatic mode2');
THIS^.Messenger.Notify('We are running automatic mode3');
THIS^._verticalPiston.Messenger.Notify('We are running automatic mode4');
THIS^._verticalPiston.Messenger.Notify('We are running automatic mode5');
THIS^._verticalPiston.Messenger.Notify('We are running automatic mode6');
THIS^._gripperPiston.Messenger.Notify('We are running automatic mode7');
THIS^._gripperPiston.Messenger.Notify('We are running automatic mode8');
THIS^._gripperPiston.Messenger.Notify('We are running automatic mode9');
THIS^.Messenger.Info('We are running automatic mode1');
THIS^.Messenger.Notify('We are running automatic mode2');
THIS^.Messenger.Notify('We are running automatic mode3');
THIS^._verticalPiston.Messenger.Notify('We are running automatic mode4');
THIS^._verticalPiston.Messenger.Notify('We are running automatic mode5');
THIS^._verticalPiston.Messenger.Notify('We are running automatic mode6');
THIS^._gripperPiston.Messenger.Notify('We are running automatic mode7');
THIS^._gripperPiston.Messenger.Notify('We are running automatic mode8');
THIS^._gripperPiston.Messenger.Notify('We are running automatic mode9');
THIS^.Messenger.Info('We are running automatic mode1');
THIS^.Messenger.Notify('We are running automatic mode2');
THIS^.Messenger.Notify('We are running automatic mode3');
THIS^._verticalPiston.Messenger.Notify('We are running automatic mode4');
THIS^._verticalPiston.Messenger.Notify('We are running automatic mode5');
THIS^._verticalPiston.Messenger.Notify('We are running automatic mode6');
THIS^._gripperPiston.Messenger.Notify('We are running automatic mode7');
THIS^._gripperPiston.Messenger.Notify('We are running automatic mode8');
THIS^._gripperPiston.Messenger.Notify('We are running automatic mode9');
THIS^.Messenger.Info('We are running automatic mode1');
THIS^.Messenger.Notify('We are running automatic mode2');
THIS^.Messenger.Notify('We are running automatic mode3');
THIS^._verticalPiston.Messenger.Notify('We are running automatic mode4');
THIS^._verticalPiston.Messenger.Notify('We are running automatic mode5');
THIS^._verticalPiston.Messenger.Notify('We are running automatic mode6');
THIS^._gripperPiston.Messenger.Notify('We are running automatic mode7');
THIS^._gripperPiston.Messenger.Notify('We are running automatic mode8');
THIS^._gripperPiston.Messenger.Notify('We are running automatic mode9');
THIS^.Messenger.Info('We are running automatic mode1');
THIS^.Messenger.Notify('We are running automatic mode2');
THIS^.Messenger.Notify('We are running automatic mode3');
THIS^._verticalPiston.Messenger.Notify('We are running automatic mode4');
THIS^._verticalPiston.Messenger.Notify('We are running automatic mode5');
THIS^._verticalPiston.Messenger.Notify('We are running automatic mode6');
THIS^._gripperPiston.Messenger.Notify('We are running automatic mode7');
THIS^._gripperPiston.Messenger.Notify('We are running automatic mode8');
THIS^._gripperPiston.Messenger.Notify('We are running automatic mode9');
THIS^.Messenger.Info('We are running automatic mode1');
THIS^.Messenger.Notify('We are running automatic mode2');
THIS^.Messenger.Notify('We are running automatic mode3');
THIS^._verticalPiston.Messenger.Notify('We are running automatic mode4');
THIS^._verticalPiston.Messenger.Notify('We are running automatic mode5');
THIS^._verticalPiston.Messenger.Notify('We are running automatic mode6');
THIS^._gripperPiston.Messenger.Notify('We are running automatic mode7');
THIS^._gripperPiston.Messenger.Notify('We are running automatic mode8');
THIS^._gripperPiston.Messenger.Notify('We are running automatic mode9');
THIS^.Messenger.Info('We are running automatic mode1');
THIS^.Messenger.Notify('We are running automatic mode2');
THIS^.Messenger.Notify('We are running automatic mode3');
THIS^._verticalPiston.Messenger.Notify('We are running automatic mode4');
THIS^._verticalPiston.Messenger.Notify('We are running automatic mode5');
THIS^._verticalPiston.Messenger.Notify('We are running automatic mode6');
THIS^._gripperPiston.Messenger.Notify('We are running automatic mode7');
THIS^._gripperPiston.Messenger.Notify('We are running automatic mode8');
THIS^._gripperPiston.Messenger.Notify('We are running automatic mode9');
THIS^.Messenger.Info('We are running automatic mode1');
THIS^.Messenger.Notify('We are running automatic mode2');
THIS^.Messenger.Notify('We are running automatic mode3');
THIS^._verticalPiston.Messenger.Notify('We are running automatic mode4');
THIS^._verticalPiston.Messenger.Notify('We are running automatic mode5');
THIS^._verticalPiston.Messenger.Notify('We are running automatic mode6');
THIS^._gripperPiston.Messenger.Notify('We are running automatic mode7');
THIS^._gripperPiston.Messenger.Notify('We are running automatic mode8');
THIS^._gripperPiston.Messenger.Notify('We are running automatic mode9');
//END_IF;
// THIS^.Context.Environment.Messaging.Resume();
_horizontalPiston();
_verticalPiston();
_gripperPiston();

IF (THIS^.State = 0) THEN
    IF (_verticalPiston.MoveUp().Done AND_THEN _horizontalPiston.MoveLeft().Done AND_THEN _gripperPiston.Open().Done) THEN
        THIS^.ChangeState(10);
    END_IF
END_IF

IF (THIS^.State = 10) THEN
    IF (_verticalPiston.MoveDown().Done) THEN
        THIS^.ChangeState(20);
    END_IF
END_IF

IF (THIS^.State = 20) THEN
    IF (_gripperPiston.Close().Done) THEN
        THIS^.ChangeState(30);
    END_IF
END_IF

IF (THIS^.State = 30) THEN
    IF (_verticalPiston.MoveUp().Done) THEN
        THIS^.ChangeState(40);
    END_IF
END_IF

IF (THIS^.State = 40) THEN
    IF (_horizontalPiston.MoveRight().Done) THEN
        THIS^.ChangeState(50);
    END_IF
END_IF

IF (THIS^.State = 50) THEN
    IF (_verticalPiston.MoveDown().Done) THEN
        THIS^.ChangeState(60);
    END_IF
END_IF

IF (THIS^.State = 60) THEN
    IF (_gripperPiston.Open().Done) THEN
        THIS^.ChangeState(0);
    END_IF
END_IF

END_FUNCTION_BLOCK

// ---- Examples/Implementation/TcoContext/TcoContext_App_1.TcPOU
FUNCTION_BLOCK TcoContext_App_1 EXTENDS TcoCore.TcoContext
VAR_INPUT
END_VAR
VAR_OUTPUT
END_VAR
VAR
    ResetToZero : BOOL := TRUE;
    C1 : LINT := 100;
    C2 : LINT := 200;
    TcoObject_Counter_1 : TcoObject_Counter(THIS^);
    TcoObject_Counter_2 : TcoObject_Counter(THIS^);
    Cycle : LINT := -1;
    TcoTask_DownCounter_1 : TcoTask_DownCounter(THIS^);
    TcoTask_DownCounter_2 : TcoTask_DownCounter(THIS^);
    TcoObject_Counter_1_CountUp_Done_RTRIG : R_TRIG;
    TcoObject_Counter_1_CountDown_Done_RTRIG : R_TRIG;
    TcoObject_Counter_2_CountUp_Done_RTRIG : R_TRIG;
    TcoObject_Counter_2_CountDown_Done_RTRIG : R_TRIG;
    TcoObject_Counter_1_CountUp_Reset : BOOL;
    TcoObject_Counter_1_CountDown_Reset : BOOL;
    TcoObject_Counter_2_CountUp_Reset : BOOL;
    TcoObject_Counter_2_CountDown_Reset : BOOL;
END_VAR

METHOD PROTECTED Main
//VAR
//	state : TcoState(THIS^,false);
//END_VAR
//TcoTaskInvokeLevel();
//TcoTaskInvokeImpulse();
TcoTaskInvokeReset();
//state.Restore(TcoObject_Counter_1.TcoTask_CountUp).Restore(TcoObject_Counter_2.TcoTask_CountUp);
TcoTaskImplementation();
END_METHOD

METHOD TcoTaskImplementation
VAR_INPUT
END_VAR
THIS^.TcoTask_DownCounter_1();

//Init Invoke
IF THIS^.TcoTask_DownCounter_1.CounterValue = -1 THEN
    THIS^.TcoTask_DownCounter_1.SetUpValue := C1;
    THIS^.TcoTask_DownCounter_1.Invoke();
END_IF

//Next Invoke during execution
IF THIS^.TcoTask_DownCounter_1.InTheMiddle THEN
    THIS^.TcoTask_DownCounter_1.SetUpValue := 2 * THIS^.TcoTask_DownCounter_1.SetUpValue;
    THIS^.TcoTask_DownCounter_1.Invoke();
END_IF

//Done and Invoke again
IF THIS^.TcoTask_DownCounter_1.Done THEN
    THIS^.TcoTask_DownCounter_1.SetUpValue := C1;
    THIS^.TcoTask_DownCounter_1.Invoke();
END_IF

THIS^.TcoTask_DownCounter_2();

//Init Invoke
IF THIS^.TcoTask_DownCounter_2.CounterValue = -1 THEN
    THIS^.TcoTask_DownCounter_2.SetUpValue := C2;
    THIS^.TcoTask_DownCounter_2.Invoke();
END_IF

//Next Invoke during execution
IF THIS^.TcoTask_DownCounter_2.InTheMiddle THEN
    THIS^.TcoTask_DownCounter_2.SetUpValue := 2 * THIS^.TcoTask_DownCounter_2.SetUpValue;
    THIS^.TcoTask_DownCounter_2.Invoke();
END_IF

//Done and Invoke again
IF THIS^.TcoTask_DownCounter_2.Done THEN
    THIS^.TcoTask_DownCounter_2.SetUpValue := C2;
    THIS^.TcoTask_DownCounter_2.Invoke();
END_IF
END_METHOD

METHOD TcoTaskInvokeImpulse
VAR_INPUT
END_VAR
TcoObject_Counter_1();
TcoObject_Counter_2();
TcoObject_Counter_1_CountUp_Done_RTRIG(CLK := THIS^.TcoObject_Counter_1.TcoTask_CountUp.Done);
TcoObject_Counter_1_CountDown_Done_RTRIG(CLK := THIS^.TcoObject_Counter_1.TcoTask_CountDown.Done);
TcoObject_Counter_2_CountUp_Done_RTRIG(CLK := THIS^.TcoObject_Counter_2.TcoTask_CountUp.Done);
TcoObject_Counter_2_CountDown_Done_RTRIG(CLK := THIS^.TcoObject_Counter_2.TcoTask_CountDown.Done);

IF ResetToZero THEN
    THIS^.TcoObject_Counter_1.TcoTask_ResetToZero.Invoke();
    THIS^.TcoObject_Counter_2.TcoTask_ResetToZero.Invoke();
    ResetToZero := FALSE;
END_IF

IF THIS^.TcoObject_Counter_1.TcoTask_ResetToZero.Done THEN
    THIS^.TcoObject_Counter_1.StartCountUp(C1);
    THIS^.TcoObject_Counter_1.TcoTask_ResetToZero.Restore(); //ResetToZeroTask has to be reseted, otherwise StartCountUp is called cyclically
END_IF;

IF THIS^.TcoObject_Counter_2.TcoTask_ResetToZero.Done THEN
    THIS^.TcoObject_Counter_2.StartCountUp(C2);
    THIS^.TcoObject_Counter_2.TcoTask_ResetToZero.Restore(); //ResetToZeroTask has to be reseted, otherwise StartCountUp is called cyclically
END_IF;

IF TcoObject_Counter_1_CountUp_Done_RTRIG.Q THEN
    THIS^.TcoObject_Counter_1.StartCountDown(-C1);
END_IF;

IF TcoObject_Counter_2_CountUp_Done_RTRIG.Q THEN
    THIS^.TcoObject_Counter_2.StartCountDown(-C2);
END_IF;

IF THIS^.TcoObject_Counter_1.TcoTask_CountDown.Done AND
    NOT THIS^.TcoObject_Counter_1.TcoTask_CountUp.Busy AND
    THIS^.TcoObject_Counter_2.TcoTask_CountDown.Done AND
    NOT THIS^.TcoObject_Counter_2.TcoTask_CountUp.Busy THEN
    THIS^.TcoObject_Counter_1.StartCountUp(C1);
    THIS^.TcoObject_Counter_2.StartCountUp(C2);
END_IF

Cycle := THIS^.TcoObject_Counter_2.Cycle;
END_METHOD

METHOD TcoTaskInvokeLevel
VAR_INPUT
END_VAR
TcoObject_Counter_1();
TcoObject_Counter_2();

IF ResetToZero THEN
    THIS^.TcoObject_Counter_1.TcoTask_ResetToZero.Invoke();
    THIS^.TcoObject_Counter_2.TcoTask_ResetToZero.Invoke();
    ResetToZero := FALSE;
END_IF

IF THIS^.TcoObject_Counter_1.TcoTask_ResetToZero.Done THEN
    THIS^.TcoObject_Counter_1.StartCountUp(C1);
    THIS^.TcoObject_Counter_1.TcoTask_ResetToZero.Restore(); //ResetToZeroTask has to be reseted, otherwise StartCountUp is called cyclically
END_IF;

IF THIS^.TcoObject_Counter_1.TcoTask_CountUp.Done THEN
    THIS^.TcoObject_Counter_1.StartCountDown(-C1);
END_IF;

IF THIS^.TcoObject_Counter_2.TcoTask_ResetToZero.Done THEN
    THIS^.TcoObject_Counter_2.StartCountUp(C2);
    THIS^.TcoObject_Counter_2.TcoTask_ResetToZero.Restore(); //ResetToZeroTask has to be reseted, otherwise StartCountUp is called cyclically
END_IF;

IF THIS^.TcoObject_Counter_2.TcoTask_CountUp.Done THEN
    THIS^.TcoObject_Counter_2.StartCountDown(-C2);
END_IF;

IF THIS^.TcoObject_Counter_1.TcoTask_CountDown.Done AND THIS^.TcoObject_Counter_2.TcoTask_CountDown.Done THEN
    THIS^.TcoObject_Counter_1.StartCountUp(C1);
    THIS^.TcoObject_Counter_2.StartCountUp(C2);
END_IF

Cycle := THIS^.TcoObject_Counter_2.Cycle;
END_METHOD

METHOD TcoTaskInvokeReset
VAR_INPUT
END_VAR
TcoObject_Counter_1();
TcoObject_Counter_2();
TcoObject_Counter_1_CountUp_Reset := FALSE;
TcoObject_Counter_1_CountDown_Reset := False;
TcoObject_Counter_2_CountUp_Reset := False;
TcoObject_Counter_2_CountDown_Reset := False;
THIS^.TcoObject_Counter_1.TcoTask_ResetToZero.Invoke();
THIS^.TcoObject_Counter_2.TcoTask_ResetToZero.Invoke();
THIS^.TcoObject_Counter_1.StartCountUp(C1);
THIS^.TcoObject_Counter_1.StartCountDown(-C1);
THIS^.TcoObject_Counter_2.StartCountUp(C2);
THIS^.TcoObject_Counter_2.StartCountDown(-C2);

IF THIS^.TcoObject_Counter_1.TcoTask_CountUp.Busy THEN
    THIS^.TcoObject_Counter_1.TcoTask_CountDown.Restore();
    TcoObject_Counter_1_CountDown_Reset := TRUE;
END_IF

IF THIS^.TcoObject_Counter_2.TcoTask_CountUp.Busy THEN
    THIS^.TcoObject_Counter_2.TcoTask_CountDown.Restore();
    TcoObject_Counter_2_CountDown_Reset := TRUE;
END_IF

IF THIS^.TcoObject_Counter_2.TcoTask_CountDown.Busy THEN
    THIS^.TcoObject_Counter_1.TcoTask_CountUp.Restore();
    TcoObject_Counter_1_CountUp_Reset := TRUE;
END_IF

IF THIS^.TcoObject_Counter_2.TcoTask_CountDown.Busy THEN
    THIS^.TcoObject_Counter_2.TcoTask_CountUp.Restore();
    TcoObject_Counter_2_CountUp_Reset := TRUE;
END_IF

Cycle := THIS^.TcoObject_Counter_2.Cycle;
END_METHOD

END_FUNCTION_BLOCK

// ---- Examples/Implementation/TcoObject/TcoObject_Counter.TcPOU
FUNCTION_BLOCK TcoObject_Counter EXTENDS TcoCore.TcoObject
VAR
    CounterValue : LINT;
    UpperLimit : LINT;
    LowerLimit : LINT;
    TcoTask_CountUp : TcoCore.TcoTask(THIS^);
    TcoTask_CountDown : TcoCore.TcoTask(THIS^);
    TcoTask_ResetToZero : TcoCore.TcoTask(THIS^);
    CountUp_InvokeTrigCounter : LINT;
    CountUp_DoneTrigCounter : LINT;
    CountDown_InvokeTrigCounter : LINT;
    CountDown_DoneTrigCounter : LINT;
    ResetToZero_InvokeTrigCounter : LINT;
    ResetToZero_DoneTrigCounter : LINT;
    CountUp_PreviousState : TcoCore.eTaskState;
    CountDown_PreviousState : TcoCore.eTaskState;
    ResetToZero_PreviousState : TcoCore.eTaskState;
    CountUp_Execute : BOOL;
    CountDown_Execute : BOOL;
    ResetToZero_Execute : BOOL;
    CountUp_Busy : BOOL;
    CountDown_Busy : BOOL;
    ResetToZero_Busy : BOOL;
    CountUp_Done : BOOL;
    CountDown_Done : BOOL;
    ResetToZero_Done : BOOL;
    Cycle : LINT;
END_VAR

CountUp_Execute := FALSE;
CountDown_Execute := FALSE;
ResetToZero_Execute := FALSE;
CountUp_Busy := FALSE;
CountDown_Busy := FALSE;
ResetToZero_Busy := FALSE;
CountUp_Done := FALSE;
CountDown_Done := FALSE;
ResetToZero_Done := FALSE;

//******************************************************************
IF (TcoTask_CountUp._taskState = eTaskState.Requested AND CountUp_PreviousState <> eTaskState.Requested) THEN
    CountUp_InvokeTrigCounter := CountUp_InvokeTrigCounter + 1;
END_IF

IF (TcoTask_CountUp.Execute()) THEN
    CountUp_Busy := TRUE;
    CounterValue := CounterValue + 1;
    TcoTask_CountUp.DoneWhen(CounterValue >= UpperLimit);
END_IF

IF (TcoTask_CountUp._taskState = eTaskState.Done AND CountUp_PreviousState <> eTaskState.Done) THEN
    CountUp_DoneTrigCounter := CountUp_DoneTrigCounter + 1;
END_IF

CountUp_Done := TcoTask_CountUp._taskState = eTaskState.Done;
CountUp_PreviousState := TcoTask_CountUp._taskState;

//******************************************************************
//******************************************************************
IF (TcoTask_CountDown._taskState = eTaskState.Requested AND CountDown_PreviousState <> eTaskState.Requested) THEN
    CountDown_InvokeTrigCounter := CountDown_InvokeTrigCounter + 1;
END_IF

IF (TcoTask_CountDown.Execute()) THEN
    CountDown_Busy := TRUE;
    CounterValue := CounterValue - 1;
    TcoTask_CountDown.DoneWhen(CounterValue <= LowerLimit);
END_IF

IF (TcoTask_CountDown._taskState = eTaskState.Done AND CountDown_PreviousState <> eTaskState.Done) THEN
    CountDown_DoneTrigCounter := CountDown_DoneTrigCounter + 1;
    Cycle := Cycle + 1;
END_IF

CountDown_Done := TcoTask_CountDown._taskState = eTaskState.Done;
CountDown_PreviousState := TcoTask_CountDown._taskState;

//******************************************************************
//******************************************************************
IF (TcoTask_ResetToZero._taskState = eTaskState.Requested AND ResetToZero_PreviousState <> eTaskState.Requested) THEN
    ResetToZero_InvokeTrigCounter := ResetToZero_InvokeTrigCounter + 1;
END_IF

IF (TcoTask_ResetToZero.Execute()) THEN
    ResetToZero_Busy := TRUE;
    TcoTask_ResetToZero.DoneWhen(TRUE);
END_IF

IF (TcoTask_ResetToZero._taskState = eTaskState.Done AND ResetToZero_PreviousState <> eTaskState.Done) THEN
    ResetToZero_DoneTrigCounter := ResetToZero_DoneTrigCounter + 1;
END_IF

ResetToZero_Done := TcoTask_ResetToZero._taskState = eTaskState.Done;
ResetToZero_PreviousState := TcoTask_ResetToZero._taskState;
//******************************************************************

METHOD Restore : BOOL
VAR_INPUT
END_VAR
TcoTask_CountUp.Restore();
TcoTask_CountDown.Restore();
CounterValue := 0;
ResetToZero_Execute := TRUE;
THIS^.TcoTask_ResetToZero.Invoke();
END_METHOD

METHOD StartCountDown
VAR_INPUT
    Value : LINT;
END_VAR
THIS^.LowerLimit := Value;
CountDown_Execute := TRUE;
TcoTask_CountDown.Invoke();
END_METHOD

METHOD StartCountUp
VAR_INPUT
    Value : LINT;
END_VAR
THIS^.UpperLimit := Value;
CountUp_Execute := TRUE;
TcoTask_CountUp.Invoke();
END_METHOD

END_FUNCTION_BLOCK

// ---- Examples/Implementation/TcoTask/TcoTask_DownCounter.TcPOU
FUNCTION_BLOCK TcoTask_DownCounter EXTENDS TcoCore.TcoTask
VAR
    _SetUpValue : LINT;
    _CounterValue : LINT := -1;
    _InvokeCounter : LINT;
    _DoneCounter : LINT;
END_VAR

IF (THIS^._taskState = eTaskState.Requested) THEN
    CounterValue := SetUpValue;
    _InvokeCounter := _InvokeCounter + 1;
END_IF;

IF (Execute()) THEN
    _CounterValue := _CounterValue - 1;
    DoneWhen(_CounterValue <= 0);
END_IF

IF (THIS^._taskState = eTaskState.Done) THEN
    _DoneCounter := _DoneCounter + 1;
END_IF;

PROPERTY CounterValue : LINT
GET
CounterValue := _CounterValue;
END_GET
SET
_CounterValue := CounterValue;
END_SET
END_PROPERTY

PROPERTY InTheMiddle : BOOL
GET
InTheMiddle := ABS(_SetUpValue - 2 * _CounterValue) < 1;
END_GET
END_PROPERTY

PROPERTY SetUpValue : LINT
GET
SetUpValue := _SetUpValue;
END_GET
SET
_SetUpValue := SetUpValue;
END_SET
END_PROPERTY

END_FUNCTION_BLOCK

// ---- Examples/Implementation/TcoState/TcoContext_App_2.TcPOU
FUNCTION_BLOCK TcoContext_App_2 EXTENDS TcoCore.TcoContext
VAR
    ResetToZero : BOOL := TRUE;
    C1 : LINT := 100;
    C2 : LINT := 200;
    TcoObject_Counter_1 : TcoObject_Counter(THIS^);
    TcoObject_Counter_2 : TcoObject_Counter(THIS^);
    TcoState_1 : TcoCore.TcoState(THIS^, TcoCore.eRestoreMode.None);
    //	TcoState_Counter_2	: TcoState(THIS^,TRUE);
END_VAR

METHOD PROTECTED Main
TcoObject_Counter_1();
TcoObject_Counter_2();

//THIS^.TcoObject_Counter_1.TcoTask_ResetToZero.Invoke();
//THIS^.TcoObject_Counter_2.TcoTask_ResetToZero.Invoke();
//THIS^.TcoObject_Counter_1.StartCountUp(C1);
//THIS^.TcoObject_Counter_1.StartCountDown(-C1);
//THIS^.TcoObject_Counter_2.StartCountUp(C2);
//THIS^.TcoObject_Counter_2.StartCountDown(-C2);
IF TcoState_1.State = 0 THEN
    THIS^.TcoObject_Counter_1.StartCountUp(C1);
    THIS^.TcoObject_Counter_2.StartCountUp(C2);
    TcoState_1.ChangeState(10);
END_IF

IF TcoState_1.State = 10 THEN
    IF THIS^.TcoObject_Counter_1.TcoTask_CountUp.Done THEN
        THIS^.TcoObject_Counter_1.StartCountDown(-C1);
        TcoState_1.ChangeState(20); //.Restore(THIS^.TcoObject_Counter_1.TcoTask_CountUp);
    END_IF
END_IF

IF TcoState_1.State = 20 THEN
    IF THIS^.TcoObject_Counter_2.TcoTask_CountUp.Done THEN
        THIS^.TcoObject_Counter_2.StartCountDown(-C2);
        TcoState_1.ChangeState(30); //.Restore(THIS^.TcoObject_Counter_2.TcoTask_CountUp);
    END_IF
END_IF

IF TcoState_1.State = 30 THEN
    IF THIS^.TcoObject_Counter_1.TcoTask_CountDown.Done AND THIS^.TcoObject_Counter_2.TcoTask_CountDown.Done THEN
        TcoState_1.ChangeState(0); //.Restore(THIS^.TcoObject_Counter_1.TcoTask_CountUp);
    END_IF
END_IF
END_METHOD

END_FUNCTION_BLOCK

// ---- Examples/Structured/StructuredObject.TcPOU
FUNCTION_BLOCK StructuredObject EXTENDS TcoCore.TcoObject

END_FUNCTION_BLOCK

// ---- Examples/WaveForm/TcoContext_Waveform.TcPOU
FUNCTION_BLOCK TcoContext_Waveform EXTENDS TcoCore._internals_TcoContext
VAR
    _TcoObject_Waveform : TcoObject_Waveform(THIS^);
END_VAR

METHOD PROTECTED Main
_TcoObject_Waveform();
END_METHOD

END_FUNCTION_BLOCK

// ---- Examples/WaveForm/TcoObject_Waveform.TcPOU
FUNCTION_BLOCK TcoObject_Waveform EXTENDS TcoObject
VAR
    _TcoTask_Waveform : TcoCore.TcoTask(THIS^);
    _TcoState_Waveform : TcoCore.TcoState(THIS^, TcoCore.eRestoreMode.None);
    _TcoState_WaveformSequence_1 : TcoState_WaveformSequence(THIS^, TcoCore.eRestoreMode.None);
    _TcoState_WaveformSequence_2 : TcoState_WaveformSequence(THIS^, TcoCore.eRestoreMode.None);
    _Value1 : LREAL;
    _Value2 : LREAL;
    _Value : LREAL;
    _X : ULINT;
    _PlcCycleOffset : ULINT;
    _PlcCycle : ULINT;
    _Reset : BOOL := TRUE;
    _Start : BOOL := TRUE;
END_VAR

IF _Reset THEN
    THIS^._TcoTask_Waveform.Restore();
    _Value := _Value1 := _Value2 := 0.0;
    _X := 0;
    _Reset := FALSE;
    RETURN;
END_IF

IF _Start THEN
    THIS^.Start();
    _Start := FALSE;
END_IF

IF THIS^._TcoTask_Waveform.Execute() THEN
    THIS^.Execute();
    THIS^._TcoTask_Waveform.DoneWhen(THIS^._TcoState_Waveform.State = 20);
END_IF

METHOD Execute
//Init both signal sequences
IF _TcoState_Waveform.State = -1 THEN
    _TcoState_WaveformSequence_1.Restore();
    _TcoState_WaveformSequence_2.Restore();
    _TcoState_WaveformSequence_1.ClearWaveFormTable();
    _TcoState_WaveformSequence_2.ClearWaveFormTable();

    _TcoState_WaveformSequence_1.AddWaveFormPoint(TransitionType := eTransitionType.Linear,
        TargetValue := 100,
        Duration := 100,
        Shape := 0.0);

    _TcoState_WaveformSequence_1.AddWaveFormPoint(TransitionType := eTransitionType.Linear,
        TargetValue := 80,
        Duration := 100,
        Shape := 0.0);

    _TcoState_WaveformSequence_1.AddWaveFormPoint(TransitionType := eTransitionType.Exponential,
        TargetValue := 100,
        Duration := 100,
        Shape := -5.0);

    _TcoState_WaveformSequence_1.AddWaveFormPoint(TransitionType := eTransitionType.S_Type,
        TargetValue := 50,
        Duration := 100,
        Shape := 3.0);

    _TcoState_WaveformSequence_1.AddWaveFormPoint(TransitionType := eTransitionType.S_Type,
        TargetValue := 120,
        Duration := 100,
        Shape := 2.0);

    _TcoState_WaveformSequence_2.AddWaveFormPoint(TransitionType := eTransitionType.Linear,
        TargetValue := 100,
        Duration := 300,
        Shape := 0.0);

    _TcoState_WaveformSequence_2.AddWaveFormPoint(TransitionType := eTransitionType.Linear,
        TargetValue := 100,
        Duration := 200,
        Shape := 0.0);

    _PlcCycleOffset := THIS^.Context.StartCycleCount - 1;
    _TcoState_Waveform.ChangeState(10);
END_IF

//Execution
IF _TcoState_Waveform.State = 10 THEN
    //	IF	_TcoState_WaveformSequence_1.RunWithAutoRestore(_Value1) AND
    //		_TcoState_WaveformSequence_2.RunWithAutoRestore(_Value2) THEN
    IF _TcoState_WaveformSequence_1.RunWithManualRestore(_Value1) AND _TcoState_WaveformSequence_2.RunWithManualRestore(_Value2) THEN
        _TcoState_Waveform.ChangeState(20);
    ELSE
        _X := _X + 1;
        _PlcCycle := THIS^.Context.StartCycleCount - _PlcCycleOffset;
    END_IF

    _Value := _Value1 + _Value2;
END_IF
END_METHOD

METHOD Start
_Value := _Value1 := _Value2 := 0.0;
_X := 0;
_TcoTask_Waveform.Restore();
_TcoState_Waveform.Restore();
_TcoTask_Waveform.Invoke();
END_METHOD

END_FUNCTION_BLOCK

// ---- Examples/WaveForm/TcoState_WaveformSequence.TcPOU
FUNCTION_BLOCK TcoState_WaveformSequence EXTENDS TcoState
VAR
    _TcoTask_Transition_1 : TcoTask_Transition(THIS^);
    _TcoTask_Transition_2 : TcoTask_Transition(THIS^);
    _WaveformPointTable : ARRAY[0..10] OF WaveformPoint;
    _WaveformPointsCount : UINT;
    _ActualTransitionNumber : UINT;
END_VAR
VAR_IN_OUT
END_VAR

METHOD AddWaveFormPoint
VAR_INPUT
    TransitionType : eTransitionType := eTransitionType.None;
    TargetValue : LREAL := 0;
    Duration : UINT := 0;
    Shape : LREAL := 0.0;
END_VAR
_WaveformPointTable[_WaveformPointsCount].TransitionType := TransitionType;
_WaveformPointTable[_WaveformPointsCount].TargetValue := TargetValue;
_WaveformPointTable[_WaveformPointsCount].Duration := Duration;
_WaveformPointTable[_WaveformPointsCount].Shape := Shape;
_WaveformPointsCount := _WaveformPointsCount + 1;
END_METHOD

ACTION CheckIfFinished:
IF _ActualTransitionNumber >= _WaveformPointsCount THEN
    THIS^.ChangeState(1110);
ELSE
    THIS^.ChangeState(THIS^.State + 10);
END_IF
END_ACTION

METHOD ClearWaveFormTable
VAR
    i : INT;
END_VAR
FOR i := 0 TO 10 DO
    _WaveformPointTable[i].TransitionType := eTransitionType.None;
    _WaveformPointTable[i].TargetValue := 0;
    _WaveformPointTable[i].Duration := 0;
    _WaveformPointTable[i].Shape := 0.0;
END_FOR

_WaveformPointsCount := 0;
_ActualTransitionNumber := 0;
END_METHOD

METHOD RunWithAutoRestore : BOOL
VAR_IN_OUT
    Value : LREAL;
END_VAR
//This  method use both _TcoTask_Transition_1 and  _TcoTask_Transition_2 tasks, one for odd, another for even transition points,  so after each Done rising edge,
//no manual restore is neccessary if each task runs at least 2 PLC cycles
RunWithAutoRestore := FALSE;

//Init
IF THIS^.State = -1 THEN
    _ActualTransitionNumber := 0;
    THIS^.ChangeState(10).RestoreObject(_TcoTask_Transition_1).RestoreObject(_TcoTask_Transition_2);
    _TcoTask_Transition_1(Value := Value); //Init reference after first download
    _TcoTask_Transition_2(Value := Value); //Init reference after first download
END_IF

// 0		*********
//Check if finished
IF THIS^.State = 10 THEN
    CheckIfFinished();
END_IF

//Start transition
IF THIS^.State = 20 THEN
    StartTransition_1();
END_IF

//Wait for transition end
IF THIS^.State = 30 THEN
    WaitForTransitionEnd_1();
END_IF

// 1		*********
//Check if finished
IF THIS^.State = 110 THEN
    CheckIfFinished();
END_IF

//Start transition
IF THIS^.State = 120 THEN
    StartTransition_2();
END_IF

//Wait for transition end
IF THIS^.State = 130 THEN
    WaitForTransitionEnd_2();
END_IF

// 2		*********
//Check if finished
IF THIS^.State = 210 THEN
    CheckIfFinished();
END_IF

//Start transition
IF THIS^.State = 220 THEN
    StartTransition_1();
END_IF

//Wait for transition end
IF THIS^.State = 230 THEN
    WaitForTransitionEnd_1();
END_IF

// 3		*********
//Check if finished
IF THIS^.State = 310 THEN
    CheckIfFinished();
END_IF

//Start transition
IF THIS^.State = 320 THEN
    StartTransition_2();
END_IF

//Wait for transition end
IF THIS^.State = 330 THEN
    WaitForTransitionEnd_2();
END_IF

// 4		*********
//Check if finished
IF THIS^.State = 410 THEN
    CheckIfFinished();
END_IF

//Start transition
IF THIS^.State = 420 THEN
    StartTransition_1();
END_IF

//Wait for transition end
IF THIS^.State = 430 THEN
    WaitForTransitionEnd_1();
END_IF

// 5		*********
//Check if finished
IF THIS^.State = 510 THEN
    CheckIfFinished();
END_IF

//Start transition
IF THIS^.State = 520 THEN
    StartTransition_2();
END_IF

//Wait for transition end
IF THIS^.State = 530 THEN
    WaitForTransitionEnd_2();
END_IF

// 6		*********
//Check if finished
IF THIS^.State = 610 THEN
    CheckIfFinished();
END_IF

//Start transition
IF THIS^.State = 620 THEN
    StartTransition_1();
END_IF

//Wait for transition end
IF THIS^.State = 630 THEN
    WaitForTransitionEnd_1();
END_IF

// 7		*********
//Check if finished
IF THIS^.State = 710 THEN
    CheckIfFinished();
END_IF

//Start transition
IF THIS^.State = 720 THEN
    StartTransition_2();
END_IF

//Wait for transition end
IF THIS^.State = 730 THEN
    WaitForTransitionEnd_2();
END_IF

// 8		*********
//Check if finished
IF THIS^.State = 810 THEN
    CheckIfFinished();
END_IF

//Start transition
IF THIS^.State = 820 THEN
    StartTransition_1();
END_IF

//Wait for transition end
IF THIS^.State = 830 THEN
    WaitForTransitionEnd_1();
END_IF

// 9		*********
//Check if finished
IF THIS^.State = 910 THEN
    CheckIfFinished();
END_IF

//Start transition
IF THIS^.State = 920 THEN
    StartTransition_2();
END_IF

//Wait for transition end
IF THIS^.State = 930 THEN
    WaitForTransitionEnd_2();
END_IF

// 10	*********
//Check if finished
IF THIS^.State = 1010 THEN
    CheckIfFinished();
END_IF

//Start transition
IF THIS^.State = 1020 THEN
    StartTransition_1();
END_IF

//Wait for transition end
IF THIS^.State = 1030 THEN
    WaitForTransitionEnd_1();
END_IF

//Finished
IF THIS^.State = 1110 THEN
    RunWithAutoRestore := TRUE;
END_IF

_TcoTask_Transition_1(Value := Value);
_TcoTask_Transition_2(Value := Value);
END_METHOD

METHOD RunWithManualRestore : BOOL
VAR_IN_OUT
    Value : LREAL;
END_VAR
//This  method use only _TcoTask_Transition_1 task, so after each Done rising edge, needs to be restored manually in order to be used again in the next State in the same PLC cycle
RunWithManualRestore := FALSE;

//Init
IF THIS^.State = -1 THEN
    _ActualTransitionNumber := 0;
    THIS^.ChangeState(10).RestoreObject(_TcoTask_Transition_1).RestoreObject(_TcoTask_Transition_2);
    _TcoTask_Transition_1(Value := Value); //Init rererence after first download
END_IF

// 0		*********
//Check if finished
IF THIS^.State = 10 THEN
    CheckIfFinished();
END_IF

//Start transition
IF THIS^.State = 20 THEN
    StartTransition_1();
END_IF

//Wait for transition end
IF THIS^.State = 30 THEN
    WaitForTransitionEnd_1_AndRestore();
END_IF

// 1		*********
//Check if finished
IF THIS^.State = 110 THEN
    CheckIfFinished();
END_IF

//Start transition
IF THIS^.State = 120 THEN
    StartTransition_1();
END_IF

//Wait for transition end
IF THIS^.State = 130 THEN
    WaitForTransitionEnd_1_AndRestore();
END_IF

// 2		*********
//Check if finished
IF THIS^.State = 210 THEN
    CheckIfFinished();
END_IF

//Start transition
IF THIS^.State = 220 THEN
    StartTransition_1();
END_IF

//Wait for transition end
IF THIS^.State = 230 THEN
    WaitForTransitionEnd_1_AndRestore();
END_IF

// 3		*********
//Check if finished
IF THIS^.State = 310 THEN
    CheckIfFinished();
END_IF

//Start transition
IF THIS^.State = 320 THEN
    StartTransition_1();
END_IF

//Wait for transition end
IF THIS^.State = 330 THEN
    WaitForTransitionEnd_1_AndRestore();
END_IF

// 4		*********
//Check if finished
IF THIS^.State = 410 THEN
    CheckIfFinished();
END_IF

//Start transition
IF THIS^.State = 420 THEN
    StartTransition_1();
END_IF

//Wait for transition end
IF THIS^.State = 430 THEN
    WaitForTransitionEnd_1_AndRestore();
END_IF

// 5		*********
//Check if finished
IF THIS^.State = 510 THEN
    CheckIfFinished();
END_IF

//Start transition
IF THIS^.State = 520 THEN
    StartTransition_1();
END_IF

//Wait for transition end
IF THIS^.State = 530 THEN
    WaitForTransitionEnd_1_AndRestore();
END_IF

// 6		*********
//Check if finished
IF THIS^.State = 610 THEN
    CheckIfFinished();
END_IF

//Start transition
IF THIS^.State = 620 THEN
    StartTransition_1();
END_IF

//Wait for transition end
IF THIS^.State = 630 THEN
    WaitForTransitionEnd_1_AndRestore();
END_IF

// 7		*********
//Check if finished
IF THIS^.State = 710 THEN
    CheckIfFinished();
END_IF

//Start transition
IF THIS^.State = 720 THEN
    StartTransition_1();
END_IF

//Wait for transition end
IF THIS^.State = 730 THEN
    WaitForTransitionEnd_1_AndRestore();
END_IF

// 8		*********
//Check if finished
IF THIS^.State = 810 THEN
    CheckIfFinished();
END_IF

//Start transition
IF THIS^.State = 820 THEN
    StartTransition_1();
END_IF

//Wait for transition end
IF THIS^.State = 830 THEN
    WaitForTransitionEnd_1_AndRestore();
END_IF

// 9		*********
//Check if finished
IF THIS^.State = 910 THEN
    CheckIfFinished();
END_IF

//Start transition
IF THIS^.State = 920 THEN
    StartTransition_1();
END_IF

//Wait for transition end
IF THIS^.State = 930 THEN
    WaitForTransitionEnd_1_AndRestore();
END_IF

// 10	*********
//Check if finished
IF THIS^.State = 1010 THEN
    CheckIfFinished();
END_IF

//Start transition
IF THIS^.State = 1020 THEN
    StartTransition_1();
END_IF

//Wait for transition end
IF THIS^.State = 1030 THEN
    WaitForTransitionEnd_1_AndRestore();
END_IF

//Finished
IF THIS^.State = 1110 THEN
    RunWithManualRestore := TRUE;
END_IF

_TcoTask_Transition_1(Value := Value);
END_METHOD

ACTION StartTransition_1:
CASE THIS^._WaveformPointTable[_ActualTransitionNumber].TransitionType OF
    eTransitionType.Linear:
        THIS^._TcoTask_Transition_1.
            StartLinear(THIS^._WaveformPointTable[_ActualTransitionNumber].TargetValue, THIS^._WaveformPointTable[_ActualTransitionNumber].Duration);

        THIS^.ChangeState(THIS^.State + 10);
    eTransitionType.Exponential:
        THIS^._TcoTask_Transition_1.StartExponential(THIS^._WaveformPointTable[_ActualTransitionNumber].TargetValue,
            THIS^._WaveformPointTable[_ActualTransitionNumber].Duration,
            THIS^._WaveformPointTable[_ActualTransitionNumber].Shape);

        THIS^.ChangeState(THIS^.State + 10);
    eTransitionType.S_Type:
        THIS^._TcoTask_Transition_1.StartStype(THIS^._WaveformPointTable[_ActualTransitionNumber].TargetValue,
            THIS^._WaveformPointTable[_ActualTransitionNumber].Duration,
            THIS^._WaveformPointTable[_ActualTransitionNumber].Shape);

        THIS^.ChangeState(THIS^.State + 10);
ELSE
    THIS^.ChangeState(1110);
END_CASE
END_ACTION

ACTION StartTransition_2:
CASE THIS^._WaveformPointTable[_ActualTransitionNumber].TransitionType OF
    eTransitionType.Linear:
        THIS^._TcoTask_Transition_2.
            StartLinear(THIS^._WaveformPointTable[_ActualTransitionNumber].TargetValue, THIS^._WaveformPointTable[_ActualTransitionNumber].Duration);

        THIS^.ChangeState(THIS^.State + 10);
    eTransitionType.Exponential:
        THIS^._TcoTask_Transition_2.StartExponential(THIS^._WaveformPointTable[_ActualTransitionNumber].TargetValue,
            THIS^._WaveformPointTable[_ActualTransitionNumber].Duration,
            THIS^._WaveformPointTable[_ActualTransitionNumber].Shape);

        THIS^.ChangeState(THIS^.State + 10);
    eTransitionType.S_Type:
        THIS^._TcoTask_Transition_2.StartStype(THIS^._WaveformPointTable[_ActualTransitionNumber].TargetValue,
            THIS^._WaveformPointTable[_ActualTransitionNumber].Duration,
            THIS^._WaveformPointTable[_ActualTransitionNumber].Shape);

        THIS^.ChangeState(THIS^.State + 10);
ELSE
    THIS^.ChangeState(1110);
END_CASE
END_ACTION

ACTION WaitForTransitionEnd_1:
IF THIS^._TcoTask_Transition_1.Done THEN
    _ActualTransitionNumber := _ActualTransitionNumber + 1;
    THIS^.ChangeState(THIS^.State + 80);
END_IF
END_ACTION

ACTION WaitForTransitionEnd_1_AndRestore:
IF THIS^._TcoTask_Transition_1.Done THEN
    _ActualTransitionNumber := _ActualTransitionNumber + 1;
    THIS^.ChangeState(THIS^.State + 80).RestoreObject(_TcoTask_Transition_1);
END_IF
END_ACTION

ACTION WaitForTransitionEnd_2:
IF THIS^._TcoTask_Transition_2.Done THEN
    _ActualTransitionNumber := _ActualTransitionNumber + 1;
    THIS^.ChangeState(THIS^.State + 80);
END_IF
END_ACTION

ACTION WaitForTransitionEnd_2_AndRestore:
IF THIS^._TcoTask_Transition_2.Done THEN
    _ActualTransitionNumber := _ActualTransitionNumber + 1;
    THIS^.ChangeState(THIS^.State + 80).RestoreObject(_TcoTask_Transition_2);
END_IF
END_ACTION

END_FUNCTION_BLOCK

// ---- Examples/WaveForm/TcoTask_Transition.TcPOU
FUNCTION_BLOCK TcoTask_Transition EXTENDS TcoCore.TcoTask
VAR
    _TransitionType : eTransitionType; //Type of transition
    _k0 : LREAL; //Linear constant
    _StartValue : LREAL; //Value before transition has been started
    _TargetValue : LREAL; //Value need to be reached after transition is finished
    _Elapsed : UINT; //Elapsed "time" (number of PLC cycles) from start of the transition
    _TransitionDuration : UINT; //Number of PLC cycles during which the "_TargetValue" must be reached
    _t0 : LREAL; //Time constant
    _x0 : LREAL; //offset
    _k1 : LREAL; //Nonlinear constant
    _k2 : LREAL; //Nonlinear constant
    _k3 : LREAL; //Nonlinear constant
    _k4 : LREAL; //Nonlinear constant
    _ImmediateChange : BOOL; //Immediate start new transition, even if previous has not yet been completed
END_VAR
VAR_IN_OUT
    Value : LREAL;
END_VAR

IF (Execute()) THEN
    _Elapsed := _Elapsed + 1;

    CASE _TransitionType OF
        eTransitionType.Linear:
            Value := _x0 + _k0 * _Elapsed;

            IF _k0 > 0 THEN
                THIS^.DoneWhen(Value >= _TargetValue);
            ELSIF _k0 < 0 THEN
                THIS^.DoneWhen(Value <= _TargetValue);
            ELSE
                THIS^.DoneWhen(_Elapsed >= _TransitionDuration);
            END_IF
        eTransitionType.Exponential:
            Value := _x0 + _k0 * EXP(_t0 * _Elapsed);

            IF _k1 > 0 THEN
                THIS^.DoneWhen(Value >= _TargetValue);
            ELSIF _k1 < 0 THEN
                THIS^.DoneWhen(Value <= _TargetValue);
            ELSE
                THIS^.DoneWhen(_Elapsed >= _TransitionDuration);
            END_IF
        eTransitionType.S_Type:
            Value := _x0 + (_k1 * EXP(_t0 * _Elapsed) + _k2) / (_k3 * EXP(_t0 * _Elapsed) + _k4);

            IF _k1 > 0 THEN
                THIS^.DoneWhen(Value >= _TargetValue);
            ELSIF _k1 < 0 THEN
                THIS^.DoneWhen(Value <= _TargetValue);
            ELSE
                THIS^.DoneWhen(_Elapsed >= _TransitionDuration);
            END_IF
    ELSE
        Value := Value;
        THIS^.DoneWhen(_Elapsed >= _TransitionDuration);
    END_CASE
END_IF

PROPERTY ImmediateChange : BOOL
GET
ImmediateChange := _ImmediateChange;
END_GET
SET
_ImmediateChange := ImmediateChange;
END_SET
END_PROPERTY

METHOD StartExponential
VAR_INPUT
    TargetValue : LREAL; //Value to be reached in "Duration" PLC cycles
    Duration : UINT; //Number of PLC cycles during which the "TargetValue" must be reached
    Shape : LREAL; //Define curve shape, 0 -linear, the higher absolute value the steeper curve, if positive - convex curve type, if negative - curve type
END_VAR
IF THIS^._taskState = eTaskState.Ready OR THIS^._taskState = eTaskState.Done OR THIS^.ImmediateChange THEN
    IF Shape = 0 THEN
        StartLinear(TargetValue, Duration);
    ELSE
        _TransitionType := eTransitionType.Exponential;
        _StartValue := Value;
        _TargetValue := TargetValue;
        _Elapsed := 0;
        _TransitionDuration := Duration;

        IF Duration = 0 THEN
            _TransitionDuration := 1;
        END_IF

        _t0 := Shape / _TransitionDuration;
        _k0 := (_TargetValue - _StartValue) / (EXP(Shape) - 1);
        _x0 := _StartValue - _k0;
        _k1 := (_TargetValue - _StartValue);
        THIS^.Invoke();
    END_IF
END_IF
END_METHOD

METHOD StartLinear
VAR_INPUT
    TargetValue : LREAL; //Value to be reached in "Duration" PLC cycles
    Duration : UINT; //Number of PLC cycles during which the "TargetValue" must be reached
END_VAR
IF THIS^._taskState = eTaskState.Ready OR THIS^._taskState = eTaskState.Done OR THIS^.ImmediateChange THEN
    _TransitionType := eTransitionType.Linear;
    _StartValue := Value;
    _TargetValue := TargetValue;
    _Elapsed := 0;
    _TransitionDuration := Duration;

    IF Duration = 0 THEN
        _TransitionDuration := 1;
    END_IF

    _x0 := _StartValue;
    _k0 := (_TargetValue - _StartValue) / _TransitionDuration;
    THIS^.Invoke();
END_IF
END_METHOD

METHOD StartStype
VAR_INPUT
    TargetValue : LREAL; //Value to be reached in "Duration" PLC cycles
    Duration : UINT; //Number of PLC cycles during which the "TargetValue" must be reached
    Shape : LREAL; //Define curve shape, 0 -linear, the higher value the steeper S-curve
END_VAR
IF THIS^._taskState = eTaskState.Ready OR THIS^._taskState = eTaskState.Done OR THIS^.ImmediateChange THEN
    IF Shape = 0 THEN
        StartLinear(TargetValue, Duration);
    ELSE
        _TransitionType := eTransitionType.S_Type;
        _StartValue := Value;
        _TargetValue := TargetValue;
        _Elapsed := 0;
        _TransitionDuration := Duration;

        IF Duration = 0 THEN
            _TransitionDuration := 1;
        END_IF

        _x0 := (_StartValue + _TargetValue) / 2;
        _k1 := (_TargetValue - _StartValue) * (1 + EXP(-2 * Shape));
        _k2 := (_TargetValue - _StartValue) * (-1 - EXP(2 * Shape));
        _k3 := 2 - 2 * EXP(-2 * Shape);
        _k4 := 2 * EXP(2 * Shape) - 2;
        _t0 := 4 * Shape / Duration;
        THIS^.Invoke();
    END_IF
END_IF
END_METHOD

END_FUNCTION_BLOCK
